	VAR robtarget OpenholeUD_4793 := [[479.2, -15.9, 180.72], [0.089899, 0.701369, 0.69888, -0.10755], [0,0,0,0], [9E9, 9E9, 9E9, 9E9, 9E9, 9E9]];
	VAR robtarget OpenholeUD_4794 := [[483.2, -15.9, 180.6], [0.102327, 0.699664, 0.696899, -0.119714], [0,0,0,0], [9E9, 9E9, 9E9, 9E9, 9E9, 9E9]];
	VAR robtarget OpenholeUD_4795 := [[487.2, -15.9, 180.48], [0.114451, 0.697783, 0.69476, -0.131563], [0,0,0,0], [9E9, 9E9, 9E9, 9E9, 9E9, 9E9]];
	VAR robtarget OpenholeUD_4796 := [[491.2, -15.9, 180.36], [0.126252, 0.695745, 0.69248, -0.143081], [0,0,0,0], [9E9, 9E9, 9E9, 9E9, 9E9, 9E9]];
	VAR robtarget OpenholeUD_4797 := [[495.19, -15.9, 180.24], [0.137713, 0.693567, 0.690077, -0.154251], [0,0,0,0], [9E9, 9E9, 9E9, 9E9, 9E9, 9E9]];
	VAR robtarget OpenholeUD_4798 := [[499.19, -15.9, 180.12], [0.148822, 0.691268, 0.687571, -0.165065], [0,0,0,0], [9E9, 9E9, 9E9, 9E9, 9E9, 9E9]];
	VAR robtarget OpenholeUD_4799 := [[503.19, -15.9, 180], [0.159571, 0.688867, 0.684978, -0.175514], [0,0,0,0], [9E9, 9E9, 9E9, 9E9, 9E9, 9E9]];
	VAR robtarget OpenholeUD_4800 := [[509.34, -15.9, 179.82], [0.183051, 0.683002, 0.683002, -0.183051], [0,0,0,0], [9E9, 9E9, 9E9, 9E9, 9E9, 9E9]];
	VAR robtarget OpenholeUD_4801 := [[513.34, -15.9, 179.8], [0.183051, 0.683002, 0.683002, -0.183051], [0,0,0,0], [9E9, 9E9, 9E9, 9E9, 9E9, 9E9]];
	VAR robtarget OpenholeUD_4802 := [[517.34, -15.9, 179.79], [0.183051, 0.683002, 0.683002, -0.183051], [0,0,0,0], [9E9, 9E9, 9E9, 9E9, 9E9, 9E9]];
	VAR robtarget OpenholeUD_4803 := [[521.34, -15.9, 179.78], [0.183051, 0.683002, 0.683002, -0.183051], [0,0,0,0], [9E9, 9E9, 9E9, 9E9, 9E9, 9E9]];
	VAR robtarget OpenholeUD_4804 := [[525.34, -15.9, 179.77], [0.183051, 0.683002, 0.683002, -0.183051], [0,0,0,0], [9E9, 9E9, 9E9, 9E9, 9E9, 9E9]];
	VAR robtarget OpenholeUD_4805 := [[529.34, -15.9, 179.75], [0.183051, 0.683002, 0.683002, -0.183051], [0,0,0,0], [9E9, 9E9, 9E9, 9E9, 9E9, 9E9]];
	VAR robtarget OpenholeUD_4806 := [[529.34, -15.9, 179.75], [0.183051, 0.683002, 0.683002, -0.183051], [0,0,0,0], [9E9, 9E9, 9E9, 9E9, 9E9, 9E9]];
	VAR robtarget OpenholeUD_4807 := [[529.34, -14.7, 179.06], [0.183051, 0.683002, 0.683002, -0.183051], [0,0,0,0], [9E9, 9E9, 9E9, 9E9, 9E9, 9E9]];
	VAR robtarget OpenholeUD_4808 := [[525.34, -14.7, 179.07], [0.183051, 0.683002, 0.683002, -0.183051], [0,0,0,0], [9E9, 9E9, 9E9, 9E9, 9E9, 9E9]];
	VAR robtarget OpenholeUD_4809 := [[521.34, -14.7, 179.09], [0.183051, 0.683002, 0.683002, -0.183051], [0,0,0,0], [9E9, 9E9, 9E9, 9E9, 9E9, 9E9]];
	VAR robtarget OpenholeUD_4810 := [[517.34, -14.7, 179.1], [0.183051, 0.683002, 0.683002, -0.183051], [0,0,0,0], [9E9, 9E9, 9E9, 9E9, 9E9, 9E9]];
	VAR robtarget OpenholeUD_4811 := [[513.34, -14.7, 179.11], [0.183051, 0.683002, 0.683002, -0.183051], [0,0,0,0], [9E9, 9E9, 9E9, 9E9, 9E9, 9E9]];
	VAR robtarget OpenholeUD_4812 := [[509.34, -14.7, 179.12], [0.183051, 0.683002, 0.683002, -0.183051], [0,0,0,0], [9E9, 9E9, 9E9, 9E9, 9E9, 9E9]];
	VAR robtarget OpenholeUD_4813 := [[505.34, -14.7, 179.29], [0.161707, 0.688368, 0.682625, -0.184452], [0,0,0,0], [9E9, 9E9, 9E9, 9E9, 9E9, 9E9]];
	VAR robtarget OpenholeUD_4814 := [[501.35, -14.7, 179.46], [0.15109, 0.690776, 0.685295, -0.174272], [0,0,0,0], [9E9, 9E9, 9E9, 9E9, 9E9, 9E9]];
	VAR robtarget OpenholeUD_4815 := [[497.35, -14.7, 179.62], [0.140112, 0.693086, 0.687891, -0.163724], [0,0,0,0], [9E9, 9E9, 9E9, 9E9, 9E9, 9E9]];
	VAR robtarget OpenholeUD_4816 := [[493.35, -14.7, 179.79], [0.12878, 0.695281, 0.690397, -0.152814], [0,0,0,0], [9E9, 9E9, 9E9, 9E9, 9E9, 9E9]];
	VAR robtarget OpenholeUD_4817 := [[489.36, -14.7, 179.96], [0.117104, 0.697343, 0.692794, -0.141548], [0,0,0,0], [9E9, 9E9, 9E9, 9E9, 9E9, 9E9]];
	VAR robtarget OpenholeUD_4818 := [[485.36, -14.7, 180.12], [0.105099, 0.699253, 0.695065, -0.129939], [0,0,0,0], [9E9, 9E9, 9E9, 9E9, 9E9, 9E9]];
	VAR robtarget OpenholeUD_4819 := [[481.36, -14.7, 180.29], [0.092784, 0.700993, 0.697191, -0.118001], [0,0,0,0], [9E9, 9E9, 9E9, 9E9, 9E9, 9E9]];
	VAR robtarget OpenholeUD_4820 := [[477.37, -14.7, 180.45], [0.08018, 0.702546, 0.699154, -0.105755], [0,0,0,0], [9E9, 9E9, 9E9, 9E9, 9E9, 9E9]];
	VAR robtarget OpenholeUD_4821 := [[473.37, -14.7, 180.62], [0.067317, 0.703895, 0.700935, -0.093223], [0,0,0,0], [9E9, 9E9, 9E9, 9E9, 9E9, 9E9]];
	VAR robtarget OpenholeUD_4822 := [[469.37, -14.7, 180.79], [0.054224, 0.705025, 0.702517, -0.080435], [0,0,0,0], [9E9, 9E9, 9E9, 9E9, 9E9, 9E9]];
	VAR robtarget OpenholeUD_4823 := [[465.38, -14.7, 180.95], [0.040937, 0.705921, 0.703885, -0.067421], [0,0,0,0], [9E9, 9E9, 9E9, 9E9, 9E9, 9E9]];
	VAR robtarget OpenholeUD_4824 := [[461.38, -14.7, 181.12], [0.027494, 0.706572, 0.705025, -0.054217], [0,0,0,0], [9E9, 9E9, 9E9, 9E9, 9E9, 9E9]];
	VAR robtarget OpenholeUD_4825 := [[454.47, -14.7, 181.41], [0.004004, 0.707095, 0.706425, -0.031051], [0,0,0,0], [9E9, 9E9, 9E9, 9E9, 9E9, 9E9]];
	VAR robtarget OpenholeUD_4826 := [[454.47, -14.7, 181.41], [0.004004, 0.707095, 0.706425, -0.031051], [0,0,0,0], [9E9, 9E9, 9E9, 9E9, 9E9, 9E9]];
	VAR robtarget OpenholeUD_4827 := [[453.25, -13.5, 181.41], [-0.004258, 0.707094, 0.706428, -0.030976], [0,0,0,0], [9E9, 9E9, 9E9, 9E9, 9E9, 9E9]];
	VAR robtarget OpenholeUD_4828 := [[457.24, -13.5, 181.2], [0.009373, 0.707045, 0.70571, -0.044424], [0,0,0,0], [9E9, 9E9, 9E9, 9E9, 9E9, 9E9]];
	VAR robtarget OpenholeUD_4829 := [[461.24, -13.5, 180.99], [0.022943, 0.706734, 0.704744, -0.057757], [0,0,0,0], [9E9, 9E9, 9E9, 9E9, 9E9, 9E9]];
	VAR robtarget OpenholeUD_4830 := [[465.23, -13.5, 180.78], [0.036407, 0.706169, 0.70354, -0.070934], [0,0,0,0], [9E9, 9E9, 9E9, 9E9, 9E9, 9E9]];
	VAR robtarget OpenholeUD_4831 := [[469.22, -13.5, 180.56], [0.049725, 0.705356, 0.70211, -0.083916], [0,0,0,0], [9E9, 9E9, 9E9, 9E9, 9E9, 9E9]];
	VAR robtarget OpenholeUD_4832 := [[473.22, -13.5, 180.35], [0.062857, 0.704307, 0.700468, -0.096668], [0,0,0,0], [9E9, 9E9, 9E9, 9E9, 9E9, 9E9]];
	VAR robtarget OpenholeUD_4833 := [[477.21, -13.5, 180.14], [0.075766, 0.703036, 0.69863, -0.109158], [0,0,0,0], [9E9, 9E9, 9E9, 9E9, 9E9, 9E9]];
	VAR robtarget OpenholeUD_4834 := [[481.21, -13.5, 179.93], [0.088422, 0.701557, 0.696615, -0.12136], [0,0,0,0], [9E9, 9E9, 9E9, 9E9, 9E9, 9E9]];
	VAR robtarget OpenholeUD_4835 := [[485.2, -13.5, 179.71], [0.100796, 0.699886, 0.694438, -0.13325], [0,0,0,0], [9E9, 9E9, 9E9, 9E9, 9E9, 9E9]];
	VAR robtarget OpenholeUD_4836 := [[489.2, -13.5, 179.5], [0.112865, 0.698041, 0.69212, -0.144808], [0,0,0,0], [9E9, 9E9, 9E9, 9E9, 9E9, 9E9]];
	VAR robtarget OpenholeUD_4837 := [[493.19, -13.5, 179.29], [0.124609, 0.696041, 0.689679, -0.15602], [0,0,0,0], [9E9, 9E9, 9E9, 9E9, 9E9, 9E9]];
	VAR robtarget OpenholeUD_4838 := [[497.18, -13.5, 179.08], [0.136013, 0.693902, 0.687134, -0.166875], [0,0,0,0], [9E9, 9E9, 9E9, 9E9, 9E9, 9E9]];
	VAR robtarget OpenholeUD_4839 := [[501.18, -13.5, 178.86], [0.147067, 0.691644, 0.684501, -0.177366], [0,0,0,0], [9E9, 9E9, 9E9, 9E9, 9E9, 9E9]];
	VAR robtarget OpenholeUD_4840 := [[505.17, -13.5, 178.65], [0.157761, 0.689283, 0.681798, -0.187488], [0,0,0,0], [9E9, 9E9, 9E9, 9E9, 9E9, 9E9]];
	VAR robtarget OpenholeUD_4841 := [[509.34, -13.5, 178.43], [0.183051, 0.683002, 0.683002, -0.183051], [0,0,0,0], [9E9, 9E9, 9E9, 9E9, 9E9, 9E9]];
	VAR robtarget OpenholeUD_4842 := [[513.34, -13.5, 178.42], [0.183051, 0.683002, 0.683002, -0.183051], [0,0,0,0], [9E9, 9E9, 9E9, 9E9, 9E9, 9E9]];
	VAR robtarget OpenholeUD_4843 := [[517.34, -13.5, 178.4], [0.183051, 0.683002, 0.683002, -0.183051], [0,0,0,0], [9E9, 9E9, 9E9, 9E9, 9E9, 9E9]];
	VAR robtarget OpenholeUD_4844 := [[521.34, -13.5, 178.39], [0.183051, 0.683002, 0.683002, -0.183051], [0,0,0,0], [9E9, 9E9, 9E9, 9E9, 9E9, 9E9]];
	VAR robtarget OpenholeUD_4845 := [[529.34, -13.5, 178.37], [0.183051, 0.683002, 0.683002, -0.183051], [0,0,0,0], [9E9, 9E9, 9E9, 9E9, 9E9, 9E9]];
	VAR robtarget OpenholeUD_4846 := [[529.34, -13.5, 178.37], [0.183051, 0.683002, 0.683002, -0.183051], [0,0,0,0], [9E9, 9E9, 9E9, 9E9, 9E9, 9E9]];
	VAR robtarget OpenholeUD_4847 := [[529.34, -12.3, 177.67], [0.183051, 0.683002, 0.683002, -0.183051], [0,0,0,0], [9E9, 9E9, 9E9, 9E9, 9E9, 9E9]];
	VAR robtarget OpenholeUD_4848 := [[525.34, -12.3, 177.69], [0.183051, 0.683002, 0.683002, -0.183051], [0,0,0,0], [9E9, 9E9, 9E9, 9E9, 9E9, 9E9]];
	VAR robtarget OpenholeUD_4849 := [[521.34, -12.3, 177.7], [0.183051, 0.683002, 0.683002, -0.183051], [0,0,0,0], [9E9, 9E9, 9E9, 9E9, 9E9, 9E9]];
	VAR robtarget OpenholeUD_4850 := [[517.34, -12.3, 177.71], [0.183051, 0.683002, 0.683002, -0.183051], [0,0,0,0], [9E9, 9E9, 9E9, 9E9, 9E9, 9E9]];
	VAR robtarget OpenholeUD_4851 := [[509.34, -12.3, 177.74], [0.183051, 0.683002, 0.683002, -0.183051], [0,0,0,0], [9E9, 9E9, 9E9, 9E9, 9E9, 9E9]];
	VAR robtarget OpenholeUD_4852 := [[505.34, -12.3, 178], [0.154707, 0.689975, 0.680721, -0.19136], [0,0,0,0], [9E9, 9E9, 9E9, 9E9, 9E9, 9E9]];
	VAR robtarget OpenholeUD_4853 := [[501.35, -12.3, 178.25], [0.143967, 0.692296, 0.683462, -0.181329], [0,0,0,0], [9E9, 9E9, 9E9, 9E9, 9E9, 9E9]];
	VAR robtarget OpenholeUD_4854 := [[497.36, -12.3, 178.51], [0.132871, 0.694511, 0.686137, -0.170928], [0,0,0,0], [9E9, 9E9, 9E9, 9E9, 9E9, 9E9]];
	VAR robtarget OpenholeUD_4855 := [[493.37, -12.3, 178.77], [0.121426, 0.696603, 0.68873, -0.16016], [0,0,0,0], [9E9, 9E9, 9E9, 9E9, 9E9, 9E9]];
	VAR robtarget OpenholeUD_4856 := [[489.38, -12.3, 179.03], [0.109644, 0.698554, 0.691223, -0.149033], [0,0,0,0], [9E9, 9E9, 9E9, 9E9, 9E9, 9E9]];
	VAR robtarget OpenholeUD_4857 := [[485.39, -12.3, 179.29], [0.09754, 0.700347, 0.693598, -0.137556], [0,0,0,0], [9E9, 9E9, 9E9, 9E9, 9E9, 9E9]];
	VAR robtarget OpenholeUD_4858 := [[481.39, -12.3, 179.55], [0.085135, 0.701963, 0.695837, -0.125744], [0,0,0,0], [9E9, 9E9, 9E9, 9E9, 9E9, 9E9]];
	VAR robtarget OpenholeUD_4859 := [[477.4, -12.3, 179.8], [0.072452, 0.703385, 0.69792, -0.113614], [0,0,0,0], [9E9, 9E9, 9E9, 9E9, 9E9, 9E9]];
	VAR robtarget OpenholeUD_4860 := [[473.41, -12.3, 180.06], [0.059519, 0.704597, 0.699829, -0.10119], [0,0,0,0], [9E9, 9E9, 9E9, 9E9, 9E9, 9E9]];
	VAR robtarget OpenholeUD_4861 := [[469.42, -12.3, 180.32], [0.046369, 0.705585, 0.701547, -0.088498], [0,0,0,0], [9E9, 9E9, 9E9, 9E9, 9E9, 9E9]];
	VAR robtarget OpenholeUD_4862 := [[465.43, -12.3, 180.58], [0.033038, 0.706335, 0.703057, -0.075569], [0,0,0,0], [9E9, 9E9, 9E9, 9E9, 9E9, 9E9]];
	VAR robtarget OpenholeUD_4863 := [[461.44, -12.3, 180.84], [0.019564, 0.706836, 0.704345, -0.062437], [0,0,0,0], [9E9, 9E9, 9E9, 9E9, 9E9, 9E9]];
	VAR robtarget OpenholeUD_4864 := [[457.44, -12.3, 181.1], [0.005991, 0.707081, 0.705397, -0.04914], [0,0,0,0], [9E9, 9E9, 9E9, 9E9, 9E9, 9E9]];
	VAR robtarget OpenholeUD_4865 := [[453.45, -12.3, 181.36], [-0.007638, 0.707066, 0.706204, -0.035718], [0,0,0,0], [9E9, 9E9, 9E9, 9E9, 9E9, 9E9]];
	VAR robtarget OpenholeUD_4866 := [[449.46, -12.3, 181.61], [-0.021278, 0.706787, 0.706758, -0.022215], [0,0,0,0], [9E9, 9E9, 9E9, 9E9, 9E9, 9E9]];
	VAR robtarget OpenholeUD_4867 := [[445.47, -12.3, 181.87], [-0.034882, 0.706246, 0.707054, -0.008673], [0,0,0,0], [9E9, 9E9, 9E9, 9E9, 9E9, 9E9]];
	VAR robtarget OpenholeUD_4868 := [[441.48, -12.3, 182.13], [-0.048405, 0.705448, 0.70709, 0.004862], [0,0,0,0], [9E9, 9E9, 9E9, 9E9, 9E9, 9E9]];
	VAR robtarget OpenholeUD_4869 := [[437.49, -12.3, 182.39], [-0.061804, 0.704401, 0.706869, 0.018346], [0,0,0,0], [9E9, 9E9, 9E9, 9E9, 9E9, 9E9]];
	VAR robtarget OpenholeUD_4870 := [[433.49, -12.3, 182.65], [-0.075036, 0.703114, 0.706394, 0.031737], [0,0,0,0], [9E9, 9E9, 9E9, 9E9, 9E9, 9E9]];
	VAR robtarget OpenholeUD_4871 := [[429.5, -12.3, 182.91], [-0.088063, 0.701602, 0.705674, 0.044994], [0,0,0,0], [9E9, 9E9, 9E9, 9E9, 9E9, 9E9]];
	VAR robtarget OpenholeUD_4872 := [[425.51, -12.3, 183.16], [-0.100848, 0.699878, 0.704718, 0.058077], [0,0,0,0], [9E9, 9E9, 9E9, 9E9, 9E9, 9E9]];
	VAR robtarget OpenholeUD_4873 := [[421.52, -12.3, 183.42], [-0.11336, 0.697961, 0.703538, 0.070951], [0,0,0,0], [9E9, 9E9, 9E9, 9E9, 9E9, 9E9]];
	VAR robtarget OpenholeUD_4874 := [[417.53, -12.3, 183.68], [-0.125573, 0.695867, 0.702149, 0.083585], [0,0,0,0], [9E9, 9E9, 9E9, 9E9, 9E9, 9E9]];
	VAR robtarget OpenholeUD_4875 := [[413.54, -12.3, 183.94], [-0.137462, 0.693617, 0.700567, 0.095951], [0,0,0,0], [9E9, 9E9, 9E9, 9E9, 9E9, 9E9]];
	VAR robtarget OpenholeUD_4876 := [[409.54, -12.3, 184.2], [-0.149009, 0.691228, 0.698807, 0.108023], [0,0,0,0], [9E9, 9E9, 9E9, 9E9, 9E9, 9E9]];
	VAR robtarget OpenholeUD_4877 := [[405.55, -12.3, 184.46], [-0.1602, 0.688721, 0.696887, 0.119783], [0,0,0,0], [9E9, 9E9, 9E9, 9E9, 9E9, 9E9]];
	VAR robtarget OpenholeUD_4878 := [[401.56, -12.3, 184.72], [-0.171025, 0.686113, 0.694826, 0.131214], [0,0,0,0], [9E9, 9E9, 9E9, 9E9, 9E9, 9E9]];
	VAR robtarget OpenholeUD_4879 := [[397.57, -12.3, 184.97], [-0.181476, 0.683423, 0.69264, 0.142304], [0,0,0,0], [9E9, 9E9, 9E9, 9E9, 9E9, 9E9]];
	VAR robtarget OpenholeUD_4880 := [[393.58, -12.3, 185.23], [-0.191552, 0.680667, 0.690346, 0.153045], [0,0,0,0], [9E9, 9E9, 9E9, 9E9, 9E9, 9E9]];
	VAR robtarget OpenholeUD_4881 := [[389.36, -12.3, 185.51], [-0.201793, 0.677702, 0.687823, 0.164011], [0,0,0,0], [9E9, 9E9, 9E9, 9E9, 9E9, 9E9]];
	VAR robtarget OpenholeUD_4882 := [[385.36, -12.3, 185.52], [-0.183051, 0.683002, 0.683002, 0.183051], [0,0,0,0], [9E9, 9E9, 9E9, 9E9, 9E9, 9E9]];
	VAR robtarget OpenholeUD_4883 := [[381.36, -12.3, 185.53], [-0.183051, 0.683002, 0.683002, 0.183051], [0,0,0,0], [9E9, 9E9, 9E9, 9E9, 9E9, 9E9]];
	VAR robtarget OpenholeUD_4884 := [[377.36, -12.3, 185.54], [-0.183051, 0.683002, 0.683002, 0.183051], [0,0,0,0], [9E9, 9E9, 9E9, 9E9, 9E9, 9E9]];
	VAR robtarget OpenholeUD_4885 := [[373.36, -12.3, 185.56], [-0.183051, 0.683002, 0.683002, 0.183051], [0,0,0,0], [9E9, 9E9, 9E9, 9E9, 9E9, 9E9]];
	VAR robtarget OpenholeUD_4886 := [[369.36, -12.3, 185.57], [-0.183051, 0.683002, 0.683002, 0.183051], [0,0,0,0], [9E9, 9E9, 9E9, 9E9, 9E9, 9E9]];
	VAR robtarget OpenholeUD_4887 := [[369.36, -12.3, 185.57], [-0.183051, 0.683002, 0.683002, 0.183051], [0,0,0,0], [9E9, 9E9, 9E9, 9E9, 9E9, 9E9]];
	VAR robtarget OpenholeUD_4888 := [[369.36, -13.5, 184.88], [-0.183051, 0.683002, 0.683002, 0.183051], [0,0,0,0], [9E9, 9E9, 9E9, 9E9, 9E9, 9E9]];
	VAR robtarget OpenholeUD_4889 := [[373.36, -13.5, 184.86], [-0.183051, 0.683002, 0.683002, 0.183051], [0,0,0,0], [9E9, 9E9, 9E9, 9E9, 9E9, 9E9]];
	VAR robtarget OpenholeUD_4890 := [[377.36, -13.5, 184.85], [-0.183051, 0.683002, 0.683002, 0.183051], [0,0,0,0], [9E9, 9E9, 9E9, 9E9, 9E9, 9E9]];
	VAR robtarget OpenholeUD_4891 := [[381.36, -13.5, 184.84], [-0.183051, 0.683002, 0.683002, 0.183051], [0,0,0,0], [9E9, 9E9, 9E9, 9E9, 9E9, 9E9]];
	VAR robtarget OpenholeUD_4892 := [[389.36, -13.5, 184.81], [-0.198402, 0.678702, 0.686998, 0.167434], [0,0,0,0], [9E9, 9E9, 9E9, 9E9, 9E9, 9E9]];
	VAR robtarget OpenholeUD_4893 := [[393.35, -13.5, 184.6], [-0.188647, 0.681478, 0.689428, 0.157129], [0,0,0,0], [9E9, 9E9, 9E9, 9E9, 9E9, 9E9]];
	VAR robtarget OpenholeUD_4894 := [[397.35, -13.5, 184.39], [-0.178516, 0.684202, 0.691771, 0.146467], [0,0,0,0], [9E9, 9E9, 9E9, 9E9, 9E9, 9E9]];
	VAR robtarget OpenholeUD_4895 := [[401.34, -13.5, 184.18], [-0.168011, 0.686857, 0.694012, 0.135454], [0,0,0,0], [9E9, 9E9, 9E9, 9E9, 9E9, 9E9]];
	VAR robtarget OpenholeUD_4896 := [[405.33, -13.5, 183.96], [-0.157134, 0.689427, 0.696132, 0.124096], [0,0,0,0], [9E9, 9E9, 9E9, 9E9, 9E9, 9E9]];
	VAR robtarget OpenholeUD_4897 := [[409.33, -13.5, 183.75], [-0.145892, 0.691893, 0.698115, 0.112405], [0,0,0,0], [9E9, 9E9, 9E9, 9E9, 9E9, 9E9]];
	VAR robtarget OpenholeUD_4898 := [[413.32, -13.5, 183.54], [-0.134296, 0.694237, 0.699943, 0.100396], [0,0,0,0], [9E9, 9E9, 9E9, 9E9, 9E9, 9E9]];
	VAR robtarget OpenholeUD_4899 := [[417.32, -13.5, 183.33], [-0.122361, 0.696439, 0.701598, 0.08809], [0,0,0,0], [9E9, 9E9, 9E9, 9E9, 9E9, 9E9]];
	VAR robtarget OpenholeUD_4900 := [[421.31, -13.5, 183.11], [-0.110106, 0.698482, 0.703064, 0.075508], [0,0,0,0], [9E9, 9E9, 9E9, 9E9, 9E9, 9E9]];
	VAR robtarget OpenholeUD_4901 := [[425.31, -13.5, 182.9], [-0.097554, 0.700345, 0.704323, 0.062679], [0,0,0,0], [9E9, 9E9, 9E9, 9E9, 9E9, 9E9]];
	VAR robtarget OpenholeUD_4902 := [[429.3, -13.5, 182.69], [-0.084733, 0.702012, 0.705363, 0.049633], [0,0,0,0], [9E9, 9E9, 9E9, 9E9, 9E9, 9E9]];
	VAR robtarget OpenholeUD_4903 := [[433.29, -13.5, 182.48], [-0.071675, 0.703465, 0.706169, 0.036405], [0,0,0,0], [9E9, 9E9, 9E9, 9E9, 9E9, 9E9]];
	VAR robtarget OpenholeUD_4904 := [[437.29, -13.5, 182.26], [-0.058416, 0.70469, 0.706731, 0.023035], [0,0,0,0], [9E9, 9E9, 9E9, 9E9, 9E9, 9E9]];
	VAR robtarget OpenholeUD_4905 := [[441.28, -13.5, 182.05], [-0.044995, 0.705674, 0.707042, 0.009561], [0,0,0,0], [9E9, 9E9, 9E9, 9E9, 9E9, 9E9]];
	VAR robtarget OpenholeUD_4906 := [[445.45, -13.5, 181.83], [-0.030877, 0.706432, 0.707092, -0.004547], [0,0,0,0], [9E9, 9E9, 9E9, 9E9, 9E9, 9E9]];
	VAR robtarget OpenholeUD_4907 := [[445.45, -13.5, 181.83], [-0.030877, 0.706432, 0.707092, -0.004547], [0,0,0,0], [9E9, 9E9, 9E9, 9E9, 9E9, 9E9]];
	VAR robtarget OpenholeUD_4908 := [[444.22, -14.7, 181.83], [-0.030953, 0.706429, 0.707097, 0.003656], [0,0,0,0], [9E9, 9E9, 9E9, 9E9, 9E9, 9E9]];
	VAR robtarget OpenholeUD_4909 := [[440.23, -14.7, 182], [-0.044489, 0.705706, 0.706898, 0.017174], [0,0,0,0], [9E9, 9E9, 9E9, 9E9, 9E9, 9E9]];
	VAR robtarget OpenholeUD_4910 := [[436.23, -14.7, 182.17], [-0.0579, 0.704732, 0.706444, 0.030612], [0,0,0,0], [9E9, 9E9, 9E9, 9E9, 9E9, 9E9]];
	VAR robtarget OpenholeUD_4911 := [[432.23, -14.7, 182.33], [-0.071146, 0.703518, 0.705741, 0.04393], [0,0,0,0], [9E9, 9E9, 9E9, 9E9, 9E9, 9E9]];
	VAR robtarget OpenholeUD_4912 := [[428.24, -14.7, 182.5], [-0.084187, 0.702077, 0.704799, 0.057088], [0,0,0,0], [9E9, 9E9, 9E9, 9E9, 9E9, 9E9]];
	VAR robtarget OpenholeUD_4913 := [[424.24, -14.7, 182.67], [-0.096988, 0.700424, 0.703629, 0.070048], [0,0,0,0], [9E9, 9E9, 9E9, 9E9, 9E9, 9E9]];
	VAR robtarget OpenholeUD_4914 := [[420.25, -14.7, 182.83], [-0.109517, 0.698574, 0.702245, 0.082777], [0,0,0,0], [9E9, 9E9, 9E9, 9E9, 9E9, 9E9]];
	VAR robtarget OpenholeUD_4915 := [[416.25, -14.7, 183], [-0.121748, 0.696547, 0.700663, 0.095245], [0,0,0,0], [9E9, 9E9, 9E9, 9E9, 9E9, 9E9]];
	VAR robtarget OpenholeUD_4916 := [[412.25, -14.7, 183.17], [-0.133657, 0.69436, 0.698899, 0.107427], [0,0,0,0], [9E9, 9E9, 9E9, 9E9, 9E9, 9E9]];
	VAR robtarget OpenholeUD_4917 := [[408.26, -14.7, 183.33], [-0.145225, 0.692033, 0.69697, 0.119301], [0,0,0,0], [9E9, 9E9, 9E9, 9E9, 9E9, 9E9]];
	VAR robtarget OpenholeUD_4918 := [[404.26, -14.7, 183.5], [-0.15644, 0.689584, 0.694895, 0.13085], [0,0,0,0], [9E9, 9E9, 9E9, 9E9, 9E9, 9E9]];
	VAR robtarget OpenholeUD_4919 := [[400.26, -14.7, 183.67], [-0.167289, 0.687033, 0.69269, 0.142058], [0,0,0,0], [9E9, 9E9, 9E9, 9E9, 9E9, 9E9]];
	VAR robtarget OpenholeUD_4920 := [[396.27, -14.7, 183.83], [-0.177767, 0.684397, 0.690374, 0.152918], [0,0,0,0], [9E9, 9E9, 9E9, 9E9, 9E9, 9E9]];
	VAR robtarget OpenholeUD_4921 := [[389.35, -14.7, 184.12], [-0.195004, 0.679686, 0.686155, 0.170856], [0,0,0,0], [9E9, 9E9, 9E9, 9E9, 9E9, 9E9]];
	VAR robtarget OpenholeUD_4922 := [[385.35, -14.7, 184.13], [-0.183051, 0.683002, 0.683002, 0.183051], [0,0,0,0], [9E9, 9E9, 9E9, 9E9, 9E9, 9E9]];
	VAR robtarget OpenholeUD_4923 := [[381.35, -14.7, 184.15], [-0.183051, 0.683002, 0.683002, 0.183051], [0,0,0,0], [9E9, 9E9, 9E9, 9E9, 9E9, 9E9]];
	VAR robtarget OpenholeUD_4924 := [[377.35, -14.7, 184.16], [-0.183051, 0.683002, 0.683002, 0.183051], [0,0,0,0], [9E9, 9E9, 9E9, 9E9, 9E9, 9E9]];
	VAR robtarget OpenholeUD_4925 := [[369.35, -14.7, 184.18], [-0.183051, 0.683002, 0.683002, 0.183051], [0,0,0,0], [9E9, 9E9, 9E9, 9E9, 9E9, 9E9]];
	VAR robtarget OpenholeUD_4926 := [[369.35, -14.7, 184.18], [-0.183051, 0.683002, 0.683002, 0.183051], [0,0,0,0], [9E9, 9E9, 9E9, 9E9, 9E9, 9E9]];
	VAR robtarget OpenholeUD_4927 := [[369.35, -15.9, 183.49], [-0.183051, 0.683002, 0.683002, 0.183051], [0,0,0,0], [9E9, 9E9, 9E9, 9E9, 9E9, 9E9]];
	VAR robtarget OpenholeUD_4928 := [[373.35, -15.9, 183.48], [-0.183051, 0.683002, 0.683002, 0.183051], [0,0,0,0], [9E9, 9E9, 9E9, 9E9, 9E9, 9E9]];
	VAR robtarget OpenholeUD_4929 := [[377.35, -15.9, 183.46], [-0.183051, 0.683002, 0.683002, 0.183051], [0,0,0,0], [9E9, 9E9, 9E9, 9E9, 9E9, 9E9]];
	VAR robtarget OpenholeUD_4930 := [[381.35, -15.9, 183.45], [-0.183051, 0.683002, 0.683002, 0.183051], [0,0,0,0], [9E9, 9E9, 9E9, 9E9, 9E9, 9E9]];
	VAR robtarget OpenholeUD_4931 := [[389.35, -15.9, 183.43], [-0.191598, 0.680654, 0.685294, 0.174276], [0,0,0,0], [9E9, 9E9, 9E9, 9E9, 9E9, 9E9]];
	VAR robtarget OpenholeUD_4932 := [[393.35, -15.9, 183.31], [-0.181693, 0.683365, 0.687802, 0.164098], [0,0,0,0], [9E9, 9E9, 9E9, 9E9, 9E9, 9E9]];
	VAR robtarget OpenholeUD_4933 := [[397.35, -15.9, 183.19], [-0.171414, 0.686016, 0.690231, 0.153561], [0,0,0,0], [9E9, 9E9, 9E9, 9E9, 9E9, 9E9]];
	VAR robtarget OpenholeUD_4934 := [[401.35, -15.9, 183.07], [-0.160762, 0.688589, 0.692565, 0.142666], [0,0,0,0], [9E9, 9E9, 9E9, 9E9, 9E9, 9E9]];
	VAR robtarget OpenholeUD_4935 := [[405.35, -15.9, 182.95], [-0.149743, 0.691069, 0.694786, 0.131423], [0,0,0,0], [9E9, 9E9, 9E9, 9E9, 9E9, 9E9]];
	VAR robtarget OpenholeUD_4936 := [[409.34, -15.9, 182.83], [-0.138364, 0.693437, 0.696878, 0.11984], [0,0,0,0], [9E9, 9E9, 9E9, 9E9, 9E9, 9E9]];
	VAR robtarget OpenholeUD_4937 := [[413.34, -15.9, 182.7], [-0.126637, 0.695675, 0.698821, 0.107932], [0,0,0,0], [9E9, 9E9, 9E9, 9E9, 9E9, 9E9]];
	VAR robtarget OpenholeUD_4938 := [[417.34, -15.9, 182.58], [-0.114578, 0.697762, 0.700599, 0.095717], [0,0,0,0], [9E9, 9E9, 9E9, 9E9, 9E9, 9E9]];
	VAR robtarget OpenholeUD_4939 := [[421.34, -15.9, 182.46], [-0.102208, 0.699681, 0.702193, 0.083217], [0,0,0,0], [9E9, 9E9, 9E9, 9E9, 9E9, 9E9]];
	VAR robtarget OpenholeUD_4940 := [[425.34, -15.9, 182.34], [-0.08955, 0.701413, 0.703588, 0.07046], [0,0,0,0], [9E9, 9E9, 9E9, 9E9, 9E9, 9E9]];
	VAR robtarget OpenholeUD_4941 := [[429.33, -15.9, 182.22], [-0.076635, 0.702942, 0.704767, 0.057474], [0,0,0,0], [9E9, 9E9, 9E9, 9E9, 9E9, 9E9]];
	VAR robtarget OpenholeUD_4942 := [[433.33, -15.9, 182.1], [-0.063495, 0.70425, 0.705718, 0.044294], [0,0,0,0], [9E9, 9E9, 9E9, 9E9, 9E9, 9E9]];
	VAR robtarget OpenholeUD_4943 := [[437.33, -15.9, 181.98], [-0.050168, 0.705325, 0.706429, 0.030958], [0,0,0,0], [9E9, 9E9, 9E9, 9E9, 9E9, 9E9]];
	VAR robtarget OpenholeUD_4944 := [[443.48, -15.9, 181.8], [-0.029392, 0.706496, 0.707033, 0.010229], [0,0,0,0], [9E9, 9E9, 9E9, 9E9, 9E9, 9E9]];
	VAR robtarget OpenholeUD_4945 := [[443.48, -15.9, 181.8], [-0.029392, 0.706496, 0.707033, 0.010229], [0,0,0,0], [9E9, 9E9, 9E9, 9E9, 9E9, 9E9]];
	VAR robtarget OpenholeUD_4946 := [[443.05, -17.1, 181.74], [-0.02678, 0.706599, 0.706931, 0.015756], [0,0,0,0], [9E9, 9E9, 9E9, 9E9, 9E9, 9E9]];
	VAR robtarget OpenholeUD_4947 := [[439.05, -17.1, 181.81], [-0.040325, 0.705956, 0.706502, 0.029235], [0,0,0,0], [9E9, 9E9, 9E9, 9E9, 9E9, 9E9]];
	VAR robtarget OpenholeUD_4948 := [[435.05, -17.1, 181.89], [-0.053748, 0.705061, 0.705822, 0.042608], [0,0,0,0], [9E9, 9E9, 9E9, 9E9, 9E9, 9E9]];
	VAR robtarget OpenholeUD_4949 := [[431.05, -17.1, 181.96], [-0.067007, 0.703925, 0.704899, 0.055835], [0,0,0,0], [9E9, 9E9, 9E9, 9E9, 9E9, 9E9]];
	VAR robtarget OpenholeUD_4950 := [[427.05, -17.1, 182.03], [-0.080063, 0.70256, 0.703744, 0.068876], [0,0,0,0], [9E9, 9E9, 9E9, 9E9, 9E9, 9E9]];
	VAR robtarget OpenholeUD_4951 := [[423.05, -17.1, 182.11], [-0.092881, 0.70098, 0.702371, 0.081698], [0,0,0,0], [9E9, 9E9, 9E9, 9E9, 9E9, 9E9]];
	VAR robtarget OpenholeUD_4952 := [[419.05, -17.1, 182.18], [-0.10543, 0.699203, 0.700795, 0.094269], [0,0,0,0], [9E9, 9E9, 9E9, 9E9, 9E9, 9E9]];
	VAR robtarget OpenholeUD_4953 := [[415.05, -17.1, 182.26], [-0.117681, 0.697245, 0.699031, 0.106561], [0,0,0,0], [9E9, 9E9, 9E9, 9E9, 9E9, 9E9]];
	VAR robtarget OpenholeUD_4954 := [[411.05, -17.1, 182.33], [-0.129613, 0.695126, 0.697098, 0.11855], [0,0,0,0], [9E9, 9E9, 9E9, 9E9, 9E9, 9E9]];
	VAR robtarget OpenholeUD_4955 := [[407.05, -17.1, 182.41], [-0.141207, 0.692864, 0.695013, 0.130218], [0,0,0,0], [9E9, 9E9, 9E9, 9E9, 9E9, 9E9]];
	VAR robtarget OpenholeUD_4956 := [[403.05, -17.1, 182.48], [-0.152448, 0.690478, 0.692794, 0.141549], [0,0,0,0], [9E9, 9E9, 9E9, 9E9, 9E9, 9E9]];
	VAR robtarget OpenholeUD_4957 := [[399.06, -17.1, 182.55], [-0.163327, 0.687986, 0.690459, 0.152532], [0,0,0,0], [9E9, 9E9, 9E9, 9E9, 9E9, 9E9]];
	VAR robtarget OpenholeUD_4958 := [[395.06, -17.1, 182.63], [-0.173837, 0.685406, 0.688026, 0.163159], [0,0,0,0], [9E9, 9E9, 9E9, 9E9, 9E9, 9E9]];
	VAR robtarget OpenholeUD_4959 := [[389.35, -17.1, 182.73], [-0.188186, 0.681606, 0.684416, 0.177694], [0,0,0,0], [9E9, 9E9, 9E9, 9E9, 9E9, 9E9]];
	VAR robtarget OpenholeUD_4960 := [[385.35, -17.1, 182.75], [-0.183051, 0.683002, 0.683002, 0.183051], [0,0,0,0], [9E9, 9E9, 9E9, 9E9, 9E9, 9E9]];
	VAR robtarget OpenholeUD_4961 := [[381.35, -17.1, 182.76], [-0.183051, 0.683002, 0.683002, 0.183051], [0,0,0,0], [9E9, 9E9, 9E9, 9E9, 9E9, 9E9]];
	VAR robtarget OpenholeUD_4962 := [[377.35, -17.1, 182.77], [-0.183051, 0.683002, 0.683002, 0.183051], [0,0,0,0], [9E9, 9E9, 9E9, 9E9, 9E9, 9E9]];
	VAR robtarget OpenholeUD_4963 := [[369.35, -17.1, 182.8], [-0.183051, 0.683002, 0.683002, 0.183051], [0,0,0,0], [9E9, 9E9, 9E9, 9E9, 9E9, 9E9]];
	VAR robtarget OpenholeUD_4964 := [[369.35, -17.1, 182.8], [-0.183051, 0.683002, 0.683002, 0.183051], [0,0,0,0], [9E9, 9E9, 9E9, 9E9, 9E9, 9E9]];
	VAR robtarget OpenholeUD_4965 := [[369.35, -18.3, 182.1], [-0.183051, 0.683002, 0.683002, 0.183051], [0,0,0,0], [9E9, 9E9, 9E9, 9E9, 9E9, 9E9]];
	VAR robtarget OpenholeUD_4966 := [[373.35, -18.3, 182.09], [-0.183051, 0.683002, 0.683002, 0.183051], [0,0,0,0], [9E9, 9E9, 9E9, 9E9, 9E9, 9E9]];
	VAR robtarget OpenholeUD_4967 := [[377.35, -18.3, 182.08], [-0.183051, 0.683002, 0.683002, 0.183051], [0,0,0,0], [9E9, 9E9, 9E9, 9E9, 9E9, 9E9]];
	VAR robtarget OpenholeUD_4968 := [[381.35, -18.3, 182.07], [-0.183051, 0.683002, 0.683002, 0.183051], [0,0,0,0], [9E9, 9E9, 9E9, 9E9, 9E9, 9E9]];
	VAR robtarget OpenholeUD_4969 := [[385.35, -18.3, 182.05], [-0.183051, 0.683002, 0.683002, 0.183051], [0,0,0,0], [9E9, 9E9, 9E9, 9E9, 9E9, 9E9]];
	VAR robtarget OpenholeUD_4970 := [[389.35, -18.3, 182.04], [-0.184767, 0.68254, 0.68352, 0.181109], [0,0,0,0], [9E9, 9E9, 9E9, 9E9, 9E9, 9E9]];
	VAR robtarget OpenholeUD_4971 := [[393.35, -18.3, 182.01], [-0.174717, 0.685182, 0.686103, 0.171065], [0,0,0,0], [9E9, 9E9, 9E9, 9E9, 9E9, 9E9]];
	VAR robtarget OpenholeUD_4972 := [[397.35, -18.3, 181.98], [-0.164295, 0.687755, 0.688614, 0.160658], [0,0,0,0], [9E9, 9E9, 9E9, 9E9, 9E9, 9E9]];
	VAR robtarget OpenholeUD_4973 := [[401.35, -18.3, 181.96], [-0.153504, 0.690244, 0.691038, 0.14989], [0,0,0,0], [9E9, 9E9, 9E9, 9E9, 9E9, 9E9]];
	VAR robtarget OpenholeUD_4974 := [[405.35, -18.3, 181.93], [-0.14235, 0.69263, 0.693356, 0.138769], [0,0,0,0], [9E9, 9E9, 9E9, 9E9, 9E9, 9E9]];
	VAR robtarget OpenholeUD_4975 := [[409.35, -18.3, 181.9], [-0.130841, 0.694896, 0.695553, 0.127302], [0,0,0,0], [9E9, 9E9, 9E9, 9E9, 9E9, 9E9]];
	VAR robtarget OpenholeUD_4976 := [[413.35, -18.3, 181.87], [-0.11899, 0.697023, 0.697609, 0.115503], [0,0,0,0], [9E9, 9E9, 9E9, 9E9, 9E9, 9E9]];
	VAR robtarget OpenholeUD_4977 := [[417.35, -18.3, 181.85], [-0.106816, 0.698992, 0.699507, 0.103389], [0,0,0,0], [9E9, 9E9, 9E9, 9E9, 9E9, 9E9]];
	VAR robtarget OpenholeUD_4978 := [[421.35, -18.3, 181.82], [-0.094339, 0.700785, 0.701229, 0.090981], [0,0,0,0], [9E9, 9E9, 9E9, 9E9, 9E9, 9E9]];
	VAR robtarget OpenholeUD_4979 := [[425.35, -18.3, 181.79], [-0.081585, 0.702384, 0.702758, 0.078305], [0,0,0,0], [9E9, 9E9, 9E9, 9E9, 9E9, 9E9]];
	VAR robtarget OpenholeUD_4980 := [[429.35, -18.3, 181.76], [-0.068586, 0.703773, 0.704077, 0.065389], [0,0,0,0], [9E9, 9E9, 9E9, 9E9, 9E9, 9E9]];
	VAR robtarget OpenholeUD_4981 := [[433.35, -18.3, 181.73], [-0.055374, 0.704935, 0.705172, 0.052266], [0,0,0,0], [9E9, 9E9, 9E9, 9E9, 9E9, 9E9]];
	VAR robtarget OpenholeUD_4982 := [[437.35, -18.3, 181.71], [-0.041988, 0.705859, 0.706032, 0.038974], [0,0,0,0], [9E9, 9E9, 9E9, 9E9, 9E9, 9E9]];
	VAR robtarget OpenholeUD_4983 := [[442.86, -18.3, 181.67], [-0.02333, 0.706722, 0.706811, 0.02045], [0,0,0,0], [9E9, 9E9, 9E9, 9E9, 9E9, 9E9]];
	VAR robtarget OpenholeUD_4984 := [[442.86, -18.3, 181.67], [-0.02333, 0.706722, 0.706811, 0.02045], [0,0,0,0], [9E9, 9E9, 9E9, 9E9, 9E9, 9E9]];
	VAR robtarget OpenholeUD_4985 := [[442.9, -19.5, 181.59], [-0.019116, 0.706848, 0.706686, 0.024384], [0,0,0,0], [9E9, 9E9, 9E9, 9E9, 9E9, 9E9]];
	VAR robtarget OpenholeUD_4986 := [[438.9, -19.5, 181.57], [-0.03269, 0.706351, 0.706094, 0.03783], [0,0,0,0], [9E9, 9E9, 9E9, 9E9, 9E9, 9E9]];
	VAR robtarget OpenholeUD_4987 := [[434.9, -19.5, 181.56], [-0.046156, 0.705599, 0.705254, 0.051155], [0,0,0,0], [9E9, 9E9, 9E9, 9E9, 9E9, 9E9]];
	VAR robtarget OpenholeUD_4988 := [[430.9, -19.5, 181.54], [-0.059469, 0.704602, 0.704176, 0.064318], [0,0,0,0], [9E9, 9E9, 9E9, 9E9, 9E9, 9E9]];
	VAR robtarget OpenholeUD_4989 := [[426.9, -19.5, 181.52], [-0.072592, 0.703371, 0.702871, 0.077282], [0,0,0,0], [9E9, 9E9, 9E9, 9E9, 9E9, 9E9]];
	VAR robtarget OpenholeUD_4990 := [[422.9, -19.5, 181.5], [-0.085487, 0.70192, 0.701354, 0.090014], [0,0,0,0], [9E9, 9E9, 9E9, 9E9, 9E9, 9E9]];
	VAR robtarget OpenholeUD_4991 := [[418.9, -19.5, 181.48], [-0.098122, 0.700266, 0.699641, 0.102482], [0,0,0,0], [9E9, 9E9, 9E9, 9E9, 9E9, 9E9]];
	VAR robtarget OpenholeUD_4992 := [[414.9, -19.5, 181.46], [-0.11047, 0.698424, 0.697749, 0.11466], [0,0,0,0], [9E9, 9E9, 9E9, 9E9, 9E9, 9E9]];
	VAR robtarget OpenholeUD_4993 := [[410.9, -19.5, 181.45], [-0.122505, 0.696414, 0.695695, 0.126527], [0,0,0,0], [9E9, 9E9, 9E9, 9E9, 9E9, 9E9]];
	VAR robtarget OpenholeUD_4994 := [[406.9, -19.5, 181.43], [-0.134209, 0.694253, 0.693497, 0.138065], [0,0,0,0], [9E9, 9E9, 9E9, 9E9, 9E9, 9E9]];
	VAR robtarget OpenholeUD_4995 := [[402.9, -19.5, 181.41], [-0.145566, 0.691961, 0.691174, 0.149259], [0,0,0,0], [9E9, 9E9, 9E9, 9E9, 9E9, 9E9]];
	VAR robtarget OpenholeUD_4996 := [[398.9, -19.5, 181.39], [-0.156566, 0.689556, 0.688744, 0.160099], [0,0,0,0], [9E9, 9E9, 9E9, 9E9, 9E9, 9E9]];
	VAR robtarget OpenholeUD_4997 := [[394.9, -19.5, 181.37], [-0.167199, 0.687055, 0.686224, 0.170579], [0,0,0,0], [9E9, 9E9, 9E9, 9E9, 9E9, 9E9]];
	VAR robtarget OpenholeUD_4998 := [[389.35, -19.5, 181.35], [-0.181344, 0.683458, 0.682607, 0.18452], [0,0,0,0], [9E9, 9E9, 9E9, 9E9, 9E9, 9E9]];
	VAR robtarget OpenholeUD_4999 := [[385.35, -19.5, 181.36], [-0.183051, 0.683002, 0.683002, 0.183051], [0,0,0,0], [9E9, 9E9, 9E9, 9E9, 9E9, 9E9]];
	VAR robtarget OpenholeUD_5000 := [[381.35, -19.5, 181.37], [-0.183051, 0.683002, 0.683002, 0.183051], [0,0,0,0], [9E9, 9E9, 9E9, 9E9, 9E9, 9E9]];
	VAR robtarget OpenholeUD_5001 := [[377.35, -19.5, 181.39], [-0.183051, 0.683002, 0.683002, 0.183051], [0,0,0,0], [9E9, 9E9, 9E9, 9E9, 9E9, 9E9]];
	VAR robtarget OpenholeUD_5002 := [[373.35, -19.5, 181.4], [-0.183051, 0.683002, 0.683002, 0.183051], [0,0,0,0], [9E9, 9E9, 9E9, 9E9, 9E9, 9E9]];
	VAR robtarget OpenholeUD_5003 := [[369.35, -19.5, 181.41], [-0.183051, 0.683002, 0.683002, 0.183051], [0,0,0,0], [9E9, 9E9, 9E9, 9E9, 9E9, 9E9]];
	VAR robtarget OpenholeUD_5004 := [[369.35, -19.5, 181.41], [-0.183051, 0.683002, 0.683002, 0.183051], [0,0,0,0], [9E9, 9E9, 9E9, 9E9, 9E9, 9E9]];
	VAR robtarget OpenholeUD_5005 := [[369.34, -20.7, 180.72], [-0.183051, 0.683002, 0.683002, 0.183051], [0,0,0,0], [9E9, 9E9, 9E9, 9E9, 9E9, 9E9]];
	VAR robtarget OpenholeUD_5006 := [[373.34, -20.7, 180.71], [-0.183051, 0.683002, 0.683002, 0.183051], [0,0,0,0], [9E9, 9E9, 9E9, 9E9, 9E9, 9E9]];
	VAR robtarget OpenholeUD_5007 := [[377.34, -20.7, 180.69], [-0.183051, 0.683002, 0.683002, 0.183051], [0,0,0,0], [9E9, 9E9, 9E9, 9E9, 9E9, 9E9]];
	VAR robtarget OpenholeUD_5008 := [[381.34, -20.7, 180.68], [-0.183051, 0.683002, 0.683002, 0.183051], [0,0,0,0], [9E9, 9E9, 9E9, 9E9, 9E9, 9E9]];
	VAR robtarget OpenholeUD_5009 := [[385.34, -20.7, 180.67], [-0.183051, 0.683002, 0.683002, 0.183051], [0,0,0,0], [9E9, 9E9, 9E9, 9E9, 9E9, 9E9]];
	VAR robtarget OpenholeUD_5010 := [[389.34, -20.7, 180.65], [-0.177916, 0.684358, 0.681677, 0.187926], [0,0,0,0], [9E9, 9E9, 9E9, 9E9, 9E9, 9E9]];
	VAR robtarget OpenholeUD_5011 := [[393.34, -20.7, 180.72], [-0.167726, 0.686926, 0.684331, 0.178021], [0,0,0,0], [9E9, 9E9, 9E9, 9E9, 9E9, 9E9]];
	VAR robtarget OpenholeUD_5012 := [[397.34, -20.7, 180.78], [-0.157168, 0.689419, 0.68692, 0.167751], [0,0,0,0], [9E9, 9E9, 9E9, 9E9, 9E9, 9E9]];
	VAR robtarget OpenholeUD_5013 := [[401.34, -20.7, 180.85], [-0.146245, 0.691818, 0.68943, 0.157118], [0,0,0,0], [9E9, 9E9, 9E9, 9E9, 9E9, 9E9]];
	VAR robtarget OpenholeUD_5014 := [[405.34, -20.7, 180.91], [-0.134962, 0.694107, 0.691843, 0.146126], [0,0,0,0], [9E9, 9E9, 9E9, 9E9, 9E9, 9E9]];
	VAR robtarget OpenholeUD_5015 := [[409.34, -20.7, 180.98], [-0.123331, 0.696268, 0.694142, 0.134783], [0,0,0,0], [9E9, 9E9, 9E9, 9E9, 9E9, 9E9]];
	VAR robtarget OpenholeUD_5016 := [[413.34, -20.7, 181.04], [-0.111366, 0.698282, 0.696309, 0.123102], [0,0,0,0], [9E9, 9E9, 9E9, 9E9, 9E9, 9E9]];
	VAR robtarget OpenholeUD_5017 := [[417.34, -20.7, 181.11], [-0.099084, 0.70013, 0.698325, 0.111098], [0,0,0,0], [9E9, 9E9, 9E9, 9E9, 9E9, 9E9]];
	VAR robtarget OpenholeUD_5018 := [[421.34, -20.7, 181.17], [-0.08651, 0.701795, 0.700172, 0.09879], [0,0,0,0], [9E9, 9E9, 9E9, 9E9, 9E9, 9E9]];
	VAR robtarget OpenholeUD_5019 := [[425.34, -20.7, 181.23], [-0.07367, 0.703259, 0.701833, 0.086204], [0,0,0,0], [9E9, 9E9, 9E9, 9E9, 9E9, 9E9]];
	VAR robtarget OpenholeUD_5020 := [[429.34, -20.7, 181.3], [-0.060595, 0.704506, 0.70329, 0.073367], [0,0,0,0], [9E9, 9E9, 9E9, 9E9, 9E9, 9E9]];
	VAR robtarget OpenholeUD_5021 := [[433.34, -20.7, 181.36], [-0.047321, 0.705522, 0.70453, 0.060311], [0,0,0,0], [9E9, 9E9, 9E9, 9E9, 9E9, 9E9]];
	VAR robtarget OpenholeUD_5022 := [[437.34, -20.7, 181.43], [-0.033887, 0.706294, 0.705538, 0.047073], [0,0,0,0], [9E9, 9E9, 9E9, 9E9, 9E9, 9E9]];
	VAR robtarget OpenholeUD_5023 := [[443.16, -20.7, 181.52], [-0.014122, 0.706966, 0.70657, 0.027547], [0,0,0,0], [9E9, 9E9, 9E9, 9E9, 9E9, 9E9]];
	VAR robtarget OpenholeUD_5024 := [[443.16, -20.7, 181.52], [-0.014122, 0.706966, 0.70657, 0.027547], [0,0,0,0], [9E9, 9E9, 9E9, 9E9, 9E9, 9E9]];
	VAR robtarget OpenholeUD_5025 := [[443.69, -21.9, 181.46], [-0.008236, 0.707059, 0.706477, 0.029827], [0,0,0,0], [9E9, 9E9, 9E9, 9E9, 9E9, 9E9]];
	VAR robtarget OpenholeUD_5026 := [[439.69, -21.9, 181.35], [-0.021848, 0.706769, 0.705782, 0.043256], [0,0,0,0], [9E9, 9E9, 9E9, 9E9, 9E9, 9E9]];
	VAR robtarget OpenholeUD_5027 := [[435.69, -21.9, 181.24], [-0.035375, 0.706221, 0.704841, 0.056559], [0,0,0,0], [9E9, 9E9, 9E9, 9E9, 9E9, 9E9]];
	VAR robtarget OpenholeUD_5028 := [[431.69, -21.9, 181.13], [-0.048772, 0.705423, 0.703664, 0.069695], [0,0,0,0], [9E9, 9E9, 9E9, 9E9, 9E9, 9E9]];
	VAR robtarget OpenholeUD_5029 := [[427.69, -21.9, 181.02], [-0.061999, 0.704384, 0.702263, 0.082626], [0,0,0,0], [9E9, 9E9, 9E9, 9E9, 9E9, 9E9]];
	VAR robtarget OpenholeUD_5030 := [[423.7, -21.9, 180.91], [-0.075018, 0.703116, 0.700653, 0.095319], [0,0,0,0], [9E9, 9E9, 9E9, 9E9, 9E9, 9E9]];
	VAR robtarget OpenholeUD_5031 := [[419.7, -21.9, 180.8], [-0.087795, 0.701635, 0.69885, 0.107744], [0,0,0,0], [9E9, 9E9, 9E9, 9E9, 9E9, 9E9]];
	VAR robtarget OpenholeUD_5032 := [[415.7, -21.9, 180.69], [-0.1003, 0.699957, 0.696872, 0.119875], [0,0,0,0], [9E9, 9E9, 9E9, 9E9, 9E9, 9E9]];
	VAR robtarget OpenholeUD_5033 := [[411.7, -21.9, 180.58], [-0.112507, 0.698099, 0.694736, 0.13169], [0,0,0,0], [9E9, 9E9, 9E9, 9E9, 9E9, 9E9]];
	VAR robtarget OpenholeUD_5034 := [[407.7, -21.9, 180.47], [-0.124394, 0.696079, 0.692461, 0.143172], [0,0,0,0], [9E9, 9E9, 9E9, 9E9, 9E9, 9E9]];
	VAR robtarget OpenholeUD_5035 := [[403.7, -21.9, 180.36], [-0.135944, 0.693916, 0.690065, 0.154307], [0,0,0,0], [9E9, 9E9, 9E9, 9E9, 9E9, 9E9]];
	VAR robtarget OpenholeUD_5036 := [[399.71, -21.9, 180.25], [-0.147143, 0.691628, 0.687566, 0.165085], [0,0,0,0], [9E9, 9E9, 9E9, 9E9, 9E9, 9E9]];
	VAR robtarget OpenholeUD_5037 := [[395.71, -21.9, 180.14], [-0.157983, 0.689233, 0.684982, 0.1755], [0,0,0,0], [9E9, 9E9, 9E9, 9E9, 9E9, 9E9]];
	VAR robtarget OpenholeUD_5038 := [[389.34, -21.9, 179.96], [-0.174484, 0.685241, 0.680731, 0.191326], [0,0,0,0], [9E9, 9E9, 9E9, 9E9, 9E9, 9E9]];
	VAR robtarget OpenholeUD_5039 := [[385.34, -21.9, 179.97], [-0.183051, 0.683002, 0.683002, 0.183051], [0,0,0,0], [9E9, 9E9, 9E9, 9E9, 9E9, 9E9]];
	VAR robtarget OpenholeUD_5040 := [[381.34, -21.9, 179.99], [-0.183051, 0.683002, 0.683002, 0.183051], [0,0,0,0], [9E9, 9E9, 9E9, 9E9, 9E9, 9E9]];
	VAR robtarget OpenholeUD_5041 := [[377.34, -21.9, 180], [-0.183051, 0.683002, 0.683002, 0.183051], [0,0,0,0], [9E9, 9E9, 9E9, 9E9, 9E9, 9E9]];
	VAR robtarget OpenholeUD_5042 := [[373.34, -21.9, 180.01], [-0.183051, 0.683002, 0.683002, 0.183051], [0,0,0,0], [9E9, 9E9, 9E9, 9E9, 9E9, 9E9]];
	VAR robtarget OpenholeUD_5043 := [[369.34, -21.9, 180.02], [-0.183051, 0.683002, 0.683002, 0.183051], [0,0,0,0], [9E9, 9E9, 9E9, 9E9, 9E9, 9E9]];
	VAR robtarget OpenholeUD_5044 := [[369.34, -21.9, 180.02], [-0.183051, 0.683002, 0.683002, 0.183051], [0,0,0,0], [9E9, 9E9, 9E9, 9E9, 9E9, 9E9]];
	VAR robtarget OpenholeUD_5045 := [[369.34, -23.1, 179.33], [-0.183051, 0.683002, 0.683002, 0.183051], [0,0,0,0], [9E9, 9E9, 9E9, 9E9, 9E9, 9E9]];
	VAR robtarget OpenholeUD_5046 := [[373.34, -23.1, 179.32], [-0.183051, 0.683002, 0.683002, 0.183051], [0,0,0,0], [9E9, 9E9, 9E9, 9E9, 9E9, 9E9]];
	VAR robtarget OpenholeUD_5047 := [[377.34, -23.1, 179.31], [-0.183051, 0.683002, 0.683002, 0.183051], [0,0,0,0], [9E9, 9E9, 9E9, 9E9, 9E9, 9E9]];
	VAR robtarget OpenholeUD_5048 := [[381.34, -23.1, 179.29], [-0.183051, 0.683002, 0.683002, 0.183051], [0,0,0,0], [9E9, 9E9, 9E9, 9E9, 9E9, 9E9]];
	VAR robtarget OpenholeUD_5049 := [[385.34, -23.1, 179.28], [-0.183051, 0.683002, 0.683002, 0.183051], [0,0,0,0], [9E9, 9E9, 9E9, 9E9, 9E9, 9E9]];
	VAR robtarget OpenholeUD_5050 := [[389.34, -23.1, 179.27], [-0.17105, 0.686106, 0.679768, 0.19472], [0,0,0,0], [9E9, 9E9, 9E9, 9E9, 9E9, 9E9]];
	VAR robtarget OpenholeUD_5051 := [[393.34, -23.1, 179.43], [-0.160728, 0.688598, 0.682488, 0.184961], [0,0,0,0], [9E9, 9E9, 9E9, 9E9, 9E9, 9E9]];
	VAR robtarget OpenholeUD_5052 := [[397.33, -23.1, 179.58], [-0.15004, 0.691005, 0.685152, 0.174834], [0,0,0,0], [9E9, 9E9, 9E9, 9E9, 9E9, 9E9]];
	VAR robtarget OpenholeUD_5053 := [[401.33, -23.1, 179.74], [-0.138991, 0.693312, 0.687744, 0.164341], [0,0,0,0], [9E9, 9E9, 9E9, 9E9, 9E9, 9E9]];
	VAR robtarget OpenholeUD_5054 := [[405.33, -23.1, 179.9], [-0.127589, 0.695501, 0.690248, 0.153486], [0,0,0,0], [9E9, 9E9, 9E9, 9E9, 9E9, 9E9]];
	VAR robtarget OpenholeUD_5055 := [[409.32, -23.1, 180.05], [-0.115844, 0.697553, 0.692646, 0.142275], [0,0,0,0], [9E9, 9E9, 9E9, 9E9, 9E9, 9E9]];
	VAR robtarget OpenholeUD_5056 := [[413.32, -23.1, 180.21], [-0.103772, 0.699451, 0.694919, 0.130719], [0,0,0,0], [9E9, 9E9, 9E9, 9E9, 9E9, 9E9]];
	VAR robtarget OpenholeUD_5057 := [[417.32, -23.1, 180.37], [-0.091393, 0.701176, 0.69705, 0.118832], [0,0,0,0], [9E9, 9E9, 9E9, 9E9, 9E9, 9E9]];
	VAR robtarget OpenholeUD_5058 := [[421.31, -23.1, 180.52], [-0.078731, 0.70271, 0.69902, 0.106634], [0,0,0,0], [9E9, 9E9, 9E9, 9E9, 9E9, 9E9]];
	VAR robtarget OpenholeUD_5059 := [[425.31, -23.1, 180.68], [-0.065814, 0.704037, 0.700811, 0.094147], [0,0,0,0], [9E9, 9E9, 9E9, 9E9, 9E9, 9E9]];
	VAR robtarget OpenholeUD_5060 := [[429.31, -23.1, 180.84], [-0.052674, 0.705142, 0.702406, 0.081398], [0,0,0,0], [9E9, 9E9, 9E9, 9E9, 9E9, 9E9]];
	VAR robtarget OpenholeUD_5061 := [[433.31, -23.1, 180.99], [-0.039348, 0.706011, 0.703789, 0.068419], [0,0,0,0], [9E9, 9E9, 9E9, 9E9, 9E9, 9E9]];
	VAR robtarget OpenholeUD_5062 := [[437.3, -23.1, 181.15], [-0.025875, 0.706633, 0.704946, 0.055243], [0,0,0,0], [9E9, 9E9, 9E9, 9E9, 9E9, 9E9]];
	VAR robtarget OpenholeUD_5063 := [[444.56, -23.1, 181.43], [-0.001167, 0.707106, 0.70643, 0.030937], [0,0,0,0], [9E9, 9E9, 9E9, 9E9, 9E9, 9E9]];
	VAR robtarget OpenholeUD_5064 := [[444.56, -23.1, 181.43], [-0.001167, 0.707106, 0.70643, 0.030937], [0,0,0,0], [9E9, 9E9, 9E9, 9E9, 9E9, 9E9]];
	VAR robtarget OpenholeUD_5065 := [[446.05, -24.3, 181.45], [0.00799, 0.707062, 0.706471, 0.029979], [0,0,0,0], [9E9, 9E9, 9E9, 9E9, 9E9, 9E9]];
	VAR robtarget OpenholeUD_5066 := [[442.05, -24.3, 181.25], [-0.005655, 0.707084, 0.705772, 0.043429], [0,0,0,0], [9E9, 9E9, 9E9, 9E9, 9E9, 9E9]];
	VAR robtarget OpenholeUD_5067 := [[438.06, -24.3, 181.05], [-0.019255, 0.706845, 0.704825, 0.056762], [0,0,0,0], [9E9, 9E9, 9E9, 9E9, 9E9, 9E9]];
	VAR robtarget OpenholeUD_5068 := [[434.06, -24.3, 180.85], [-0.032766, 0.706347, 0.70364, 0.069938], [0,0,0,0], [9E9, 9E9, 9E9, 9E9, 9E9, 9E9]];
	VAR robtarget OpenholeUD_5069 := [[430.07, -24.3, 180.64], [-0.046146, 0.705599, 0.702228, 0.082919], [0,0,0,0], [9E9, 9E9, 9E9, 9E9, 9E9, 9E9]];
	VAR robtarget OpenholeUD_5070 := [[426.07, -24.3, 180.44], [-0.059352, 0.704611, 0.700605, 0.095669], [0,0,0,0], [9E9, 9E9, 9E9, 9E9, 9E9, 9E9]];
	VAR robtarget OpenholeUD_5071 := [[422.08, -24.3, 180.24], [-0.072349, 0.703396, 0.698786, 0.108157], [0,0,0,0], [9E9, 9E9, 9E9, 9E9, 9E9, 9E9]];
	VAR robtarget OpenholeUD_5072 := [[418.08, -24.3, 180.03], [-0.085103, 0.701967, 0.696789, 0.120357], [0,0,0,0], [9E9, 9E9, 9E9, 9E9, 9E9, 9E9]];
	VAR robtarget OpenholeUD_5073 := [[414.09, -24.3, 179.83], [-0.097584, 0.700341, 0.69463, 0.132245], [0,0,0,0], [9E9, 9E9, 9E9, 9E9, 9E9, 9E9]];
	VAR robtarget OpenholeUD_5074 := [[410.09, -24.3, 179.63], [-0.109766, 0.698535, 0.69233, 0.143802], [0,0,0,0], [9E9, 9E9, 9E9, 9E9, 9E9, 9E9]];
	VAR robtarget OpenholeUD_5075 := [[406.1, -24.3, 179.43], [-0.121629, 0.696568, 0.689906, 0.155014], [0,0,0,0], [9E9, 9E9, 9E9, 9E9, 9E9, 9E9]];
	VAR robtarget OpenholeUD_5076 := [[402.1, -24.3, 179.22], [-0.133156, 0.694456, 0.687377, 0.165869], [0,0,0,0], [9E9, 9E9, 9E9, 9E9, 9E9, 9E9]];
	VAR robtarget OpenholeUD_5077 := [[398.11, -24.3, 179.02], [-0.144334, 0.692219, 0.68476, 0.176361], [0,0,0,0], [9E9, 9E9, 9E9, 9E9, 9E9, 9E9]];
	VAR robtarget OpenholeUD_5078 := [[394.11, -24.3, 178.82], [-0.155155, 0.689875, 0.682073, 0.186486], [0,0,0,0], [9E9, 9E9, 9E9, 9E9, 9E9, 9E9]];
	VAR robtarget OpenholeUD_5079 := [[389.34, -24.3, 178.58], [-0.167613, 0.686954, 0.678788, 0.198107], [0,0,0,0], [9E9, 9E9, 9E9, 9E9, 9E9, 9E9]];
	VAR robtarget OpenholeUD_5080 := [[385.34, -24.3, 178.59], [-0.183051, 0.683002, 0.683002, 0.183051], [0,0,0,0], [9E9, 9E9, 9E9, 9E9, 9E9, 9E9]];
	VAR robtarget OpenholeUD_5081 := [[381.34, -24.3, 178.6], [-0.183051, 0.683002, 0.683002, 0.183051], [0,0,0,0], [9E9, 9E9, 9E9, 9E9, 9E9, 9E9]];
	VAR robtarget OpenholeUD_5082 := [[377.34, -24.3, 178.61], [-0.183051, 0.683002, 0.683002, 0.183051], [0,0,0,0], [9E9, 9E9, 9E9, 9E9, 9E9, 9E9]];
	VAR robtarget OpenholeUD_5083 := [[369.34, -24.3, 178.64], [-0.183051, 0.683002, 0.683002, 0.183051], [0,0,0,0], [9E9, 9E9, 9E9, 9E9, 9E9, 9E9]];
	VAR robtarget OpenholeUD_5084 := [[369.34, -24.3, 178.64], [-0.183051, 0.683002, 0.683002, 0.183051], [0,0,0,0], [9E9, 9E9, 9E9, 9E9, 9E9, 9E9]];
	VAR robtarget OpenholeUD_5085 := [[369.34, -25.5, 177.95], [-0.183051, 0.683002, 0.683002, 0.183051], [0,0,0,0], [9E9, 9E9, 9E9, 9E9, 9E9, 9E9]];
	VAR robtarget OpenholeUD_5086 := [[373.34, -25.5, 177.93], [-0.183051, 0.683002, 0.683002, 0.183051], [0,0,0,0], [9E9, 9E9, 9E9, 9E9, 9E9, 9E9]];
	VAR robtarget OpenholeUD_5087 := [[377.34, -25.5, 177.92], [-0.183051, 0.683002, 0.683002, 0.183051], [0,0,0,0], [9E9, 9E9, 9E9, 9E9, 9E9, 9E9]];
	VAR robtarget OpenholeUD_5088 := [[381.34, -25.5, 177.91], [-0.183051, 0.683002, 0.683002, 0.183051], [0,0,0,0], [9E9, 9E9, 9E9, 9E9, 9E9, 9E9]];
	VAR robtarget OpenholeUD_5089 := [[385.34, -25.5, 177.9], [-0.183051, 0.683002, 0.683002, 0.183051], [0,0,0,0], [9E9, 9E9, 9E9, 9E9, 9E9, 9E9]];
	VAR robtarget OpenholeUD_5090 := [[389.34, -25.5, 177.88], [-0.164176, 0.687784, 0.677793, 0.201487], [0,0,0,0], [9E9, 9E9, 9E9, 9E9, 9E9, 9E9]];
	VAR robtarget OpenholeUD_5091 := [[393.33, -25.5, 178.13], [-0.153728, 0.690194, 0.680576, 0.191877], [0,0,0,0], [9E9, 9E9, 9E9, 9E9, 9E9, 9E9]];
	VAR robtarget OpenholeUD_5092 := [[397.32, -25.5, 178.38], [-0.142918, 0.692513, 0.68331, 0.1819], [0,0,0,0], [9E9, 9E9, 9E9, 9E9, 9E9, 9E9]];
	VAR robtarget OpenholeUD_5093 := [[401.31, -25.5, 178.63], [-0.131752, 0.694724, 0.685981, 0.171553], [0,0,0,0], [9E9, 9E9, 9E9, 9E9, 9E9, 9E9]];
	VAR robtarget OpenholeUD_5094 := [[405.3, -25.5, 178.88], [-0.120237, 0.696809, 0.688571, 0.16084], [0,0,0,0], [9E9, 9E9, 9E9, 9E9, 9E9, 9E9]];
	VAR robtarget OpenholeUD_5095 := [[409.3, -25.5, 179.13], [-0.108387, 0.69875, 0.691064, 0.149767], [0,0,0,0], [9E9, 9E9, 9E9, 9E9, 9E9, 9E9]];
	VAR robtarget OpenholeUD_5096 := [[413.29, -25.5, 179.38], [-0.096218, 0.70053, 0.693441, 0.138344], [0,0,0,0], [9E9, 9E9, 9E9, 9E9, 9E9, 9E9]];
	VAR robtarget OpenholeUD_5097 := [[417.28, -25.5, 179.62], [-0.083751, 0.702129, 0.695684, 0.126583], [0,0,0,0], [9E9, 9E9, 9E9, 9E9, 9E9, 9E9]];
	VAR robtarget OpenholeUD_5098 := [[421.27, -25.5, 179.87], [-0.071011, 0.703532, 0.697774, 0.114502], [0,0,0,0], [9E9, 9E9, 9E9, 9E9, 9E9, 9E9]];
	VAR robtarget OpenholeUD_5099 := [[425.27, -25.5, 180.12], [-0.058027, 0.704722, 0.699693, 0.102123], [0,0,0,0], [9E9, 9E9, 9E9, 9E9, 9E9, 9E9]];
	VAR robtarget OpenholeUD_5100 := [[429.26, -25.5, 180.37], [-0.044832, 0.705684, 0.701423, 0.089472], [0,0,0,0], [9E9, 9E9, 9E9, 9E9, 9E9, 9E9]];
	VAR robtarget OpenholeUD_5101 := [[433.25, -25.5, 180.62], [-0.031463, 0.706406, 0.702948, 0.076578], [0,0,0,0], [9E9, 9E9, 9E9, 9E9, 9E9, 9E9]];
	VAR robtarget OpenholeUD_5102 := [[437.24, -25.5, 180.87], [-0.017962, 0.706879, 0.704252, 0.063475], [0,0,0,0], [9E9, 9E9, 9E9, 9E9, 9E9, 9E9]];
	VAR robtarget OpenholeUD_5103 := [[441.23, -25.5, 181.12], [-0.004369, 0.707093, 0.705323, 0.0502], [0,0,0,0], [9E9, 9E9, 9E9, 9E9, 9E9, 9E9]];
	VAR robtarget OpenholeUD_5104 := [[445.23, -25.5, 181.36], [0.00927, 0.707046, 0.706149, 0.036793], [0,0,0,0], [9E9, 9E9, 9E9, 9E9, 9E9, 9E9]];
	VAR robtarget OpenholeUD_5105 := [[449.22, -25.5, 181.61], [0.022909, 0.706736, 0.706723, 0.023296], [0,0,0,0], [9E9, 9E9, 9E9, 9E9, 9E9, 9E9]];
	VAR robtarget OpenholeUD_5106 := [[453.21, -25.5, 181.86], [0.036502, 0.706164, 0.70704, 0.009753], [0,0,0,0], [9E9, 9E9, 9E9, 9E9, 9E9, 9E9]];
	VAR robtarget OpenholeUD_5107 := [[457.2, -25.5, 182.11], [0.050006, 0.705336, 0.707097, -0.003791], [0,0,0,0], [9E9, 9E9, 9E9, 9E9, 9E9, 9E9]];
	VAR robtarget OpenholeUD_5108 := [[461.2, -25.5, 182.36], [0.063375, 0.704261, 0.706895, -0.017293], [0,0,0,0], [9E9, 9E9, 9E9, 9E9, 9E9, 9E9]];
	VAR robtarget OpenholeUD_5109 := [[465.19, -25.5, 182.61], [0.076569, 0.702949, 0.70644, -0.030708], [0,0,0,0], [9E9, 9E9, 9E9, 9E9, 9E9, 9E9]];
	VAR robtarget OpenholeUD_5110 := [[469.18, -25.5, 182.86], [0.089549, 0.701414, 0.705737, -0.043996], [0,0,0,0], [9E9, 9E9, 9E9, 9E9, 9E9, 9E9]];
	VAR robtarget OpenholeUD_5111 := [[473.17, -25.5, 183.11], [0.102282, 0.69967, 0.704796, -0.057117], [0,0,0,0], [9E9, 9E9, 9E9, 9E9, 9E9, 9E9]];
	VAR robtarget OpenholeUD_5112 := [[477.16, -25.5, 183.35], [0.114736, 0.697736, 0.70363, -0.070034], [0,0,0,0], [9E9, 9E9, 9E9, 9E9, 9E9, 9E9]];
	VAR robtarget OpenholeUD_5113 := [[481.16, -25.5, 183.6], [0.126886, 0.695629, 0.702252, -0.082715], [0,0,0,0], [9E9, 9E9, 9E9, 9E9, 9E9, 9E9]];
	VAR robtarget OpenholeUD_5114 := [[485.15, -25.5, 183.85], [0.138709, 0.693369, 0.700678, -0.09513], [0,0,0,0], [9E9, 9E9, 9E9, 9E9, 9E9, 9E9]];
	VAR robtarget OpenholeUD_5115 := [[489.14, -25.5, 184.1], [0.150187, 0.690973, 0.698925, -0.107256], [0,0,0,0], [9E9, 9E9, 9E9, 9E9, 9E9, 9E9]];
	VAR robtarget OpenholeUD_5116 := [[493.13, -25.5, 184.35], [0.161308, 0.688462, 0.697009, -0.119071], [0,0,0,0], [9E9, 9E9, 9E9, 9E9, 9E9, 9E9]];
	VAR robtarget OpenholeUD_5117 := [[497.13, -25.5, 184.6], [0.172062, 0.685853, 0.694949, -0.130558], [0,0,0,0], [9E9, 9E9, 9E9, 9E9, 9E9, 9E9]];
	VAR robtarget OpenholeUD_5118 := [[501.12, -25.5, 184.85], [0.182444, 0.683165, 0.692763, -0.141704], [0,0,0,0], [9E9, 9E9, 9E9, 9E9, 9E9, 9E9]];
	VAR robtarget OpenholeUD_5119 := [[505.11, -25.5, 185.1], [0.192451, 0.680414, 0.690466, -0.1525], [0,0,0,0], [9E9, 9E9, 9E9, 9E9, 9E9, 9E9]];
	VAR robtarget OpenholeUD_5120 := [[509.36, -25.5, 185.36], [0.183051, 0.683002, 0.683002, -0.183051], [0,0,0,0], [9E9, 9E9, 9E9, 9E9, 9E9, 9E9]];
	VAR robtarget OpenholeUD_5121 := [[513.36, -25.5, 185.35], [0.183051, 0.683002, 0.683002, -0.183051], [0,0,0,0], [9E9, 9E9, 9E9, 9E9, 9E9, 9E9]];
	VAR robtarget OpenholeUD_5122 := [[517.36, -25.5, 185.33], [0.183051, 0.683002, 0.683002, -0.183051], [0,0,0,0], [9E9, 9E9, 9E9, 9E9, 9E9, 9E9]];
	VAR robtarget OpenholeUD_5123 := [[521.36, -25.5, 185.32], [0.183051, 0.683002, 0.683002, -0.183051], [0,0,0,0], [9E9, 9E9, 9E9, 9E9, 9E9, 9E9]];
	VAR robtarget OpenholeUD_5124 := [[529.36, -25.5, 185.3], [0.183051, 0.683002, 0.683002, -0.183051], [0,0,0,0], [9E9, 9E9, 9E9, 9E9, 9E9, 9E9]];
	VAR robtarget OpenholeUD_5125 := [[529.36, -25.5, 185.3], [0.183051, 0.683002, 0.683002, -0.183051], [0,0,0,0], [9E9, 9E9, 9E9, 9E9, 9E9, 9E9]];
	VAR robtarget OpenholeUD_5126 := [[529.36, -26.7, 185.99], [0.183051, 0.683002, 0.683002, -0.183051], [0,0,0,0], [9E9, 9E9, 9E9, 9E9, 9E9, 9E9]];
	VAR robtarget OpenholeUD_5127 := [[525.36, -26.7, 186], [0.183051, 0.683002, 0.683002, -0.183051], [0,0,0,0], [9E9, 9E9, 9E9, 9E9, 9E9, 9E9]];
	VAR robtarget OpenholeUD_5128 := [[521.36, -26.7, 186.02], [0.183051, 0.683002, 0.683002, -0.183051], [0,0,0,0], [9E9, 9E9, 9E9, 9E9, 9E9, 9E9]];
	VAR robtarget OpenholeUD_5129 := [[517.36, -26.7, 186.03], [0.183051, 0.683002, 0.683002, -0.183051], [0,0,0,0], [9E9, 9E9, 9E9, 9E9, 9E9, 9E9]];
	VAR robtarget OpenholeUD_5130 := [[509.36, -26.7, 186.05], [0.183051, 0.683002, 0.683002, -0.183051], [0,0,0,0], [9E9, 9E9, 9E9, 9E9, 9E9, 9E9]];
	VAR robtarget OpenholeUD_5131 := [[505.37, -26.7, 185.76], [0.196536, 0.679245, 0.691078, -0.149705], [0,0,0,0], [9E9, 9E9, 9E9, 9E9, 9E9, 9E9]];
	VAR robtarget OpenholeUD_5132 := [[501.38, -26.7, 185.46], [0.186631, 0.682033, 0.693335, -0.138874], [0,0,0,0], [9E9, 9E9, 9E9, 9E9, 9E9, 9E9]];
	VAR robtarget OpenholeUD_5133 := [[497.39, -26.7, 185.17], [0.17635, 0.684763, 0.695481, -0.127696], [0,0,0,0], [9E9, 9E9, 9E9, 9E9, 9E9, 9E9]];
	VAR robtarget OpenholeUD_5134 := [[493.4, -26.7, 184.87], [0.165695, 0.687419, 0.697497, -0.116179], [0,0,0,0], [9E9, 9E9, 9E9, 9E9, 9E9, 9E9]];
	VAR robtarget OpenholeUD_5135 := [[489.42, -26.7, 184.58], [0.15467, 0.689983, 0.699367, -0.104336], [0,0,0,0], [9E9, 9E9, 9E9, 9E9, 9E9, 9E9]];
	VAR robtarget OpenholeUD_5136 := [[485.43, -26.7, 184.29], [0.143285, 0.692437, 0.701072, -0.092186], [0,0,0,0], [9E9, 9E9, 9E9, 9E9, 9E9, 9E9]];
	VAR robtarget OpenholeUD_5137 := [[481.44, -26.7, 183.99], [0.131551, 0.694762, 0.702595, -0.079748], [0,0,0,0], [9E9, 9E9, 9E9, 9E9, 9E9, 9E9]];
	VAR robtarget OpenholeUD_5138 := [[477.45, -26.7, 183.7], [0.119485, 0.696939, 0.703921, -0.067049], [0,0,0,0], [9E9, 9E9, 9E9, 9E9, 9E9, 9E9]];
	VAR robtarget OpenholeUD_5139 := [[473.46, -26.7, 183.4], [0.107108, 0.698948, 0.705033, -0.054116], [0,0,0,0], [9E9, 9E9, 9E9, 9E9, 9E9, 9E9]];
	VAR robtarget OpenholeUD_5140 := [[469.47, -26.7, 183.11], [0.094446, 0.700771, 0.705918, -0.040984], [0,0,0,0], [9E9, 9E9, 9E9, 9E9, 9E9, 9E9]];
	VAR robtarget OpenholeUD_5141 := [[465.48, -26.7, 182.81], [0.081528, 0.702391, 0.706564, -0.027689], [0,0,0,0], [9E9, 9E9, 9E9, 9E9, 9E9, 9E9]];
	VAR robtarget OpenholeUD_5142 := [[461.49, -26.7, 182.52], [0.068388, 0.703792, 0.706963, -0.014269], [0,0,0,0], [9E9, 9E9, 9E9, 9E9, 9E9, 9E9]];
	VAR robtarget OpenholeUD_5143 := [[457.5, -26.7, 182.22], [0.055063, 0.70496, 0.707106, -0.000768], [0,0,0,0], [9E9, 9E9, 9E9, 9E9, 9E9, 9E9]];
	VAR robtarget OpenholeUD_5144 := [[453.51, -26.7, 181.93], [0.041595, 0.705882, 0.706991, 0.012773], [0,0,0,0], [9E9, 9E9, 9E9, 9E9, 9E9, 9E9]];
	VAR robtarget OpenholeUD_5145 := [[449.52, -26.7, 181.63], [0.028025, 0.706551, 0.706617, 0.026308], [0,0,0,0], [9E9, 9E9, 9E9, 9E9, 9E9, 9E9]];
	VAR robtarget OpenholeUD_5146 := [[445.54, -26.7, 181.34], [0.014398, 0.70696, 0.705986, 0.039793], [0,0,0,0], [9E9, 9E9, 9E9, 9E9, 9E9, 9E9]];
	VAR robtarget OpenholeUD_5147 := [[441.55, -26.7, 181.05], [0.000761, 0.707106, 0.705104, 0.053185], [0,0,0,0], [9E9, 9E9, 9E9, 9E9, 9E9, 9E9]];
	VAR robtarget OpenholeUD_5148 := [[437.56, -26.7, 180.75], [-0.01284, 0.70699, 0.703978, 0.066441], [0,0,0,0], [9E9, 9E9, 9E9, 9E9, 9E9, 9E9]];
	VAR robtarget OpenholeUD_5149 := [[433.57, -26.7, 180.46], [-0.026362, 0.706615, 0.702621, 0.079522], [0,0,0,0], [9E9, 9E9, 9E9, 9E9, 9E9, 9E9]];
	VAR robtarget OpenholeUD_5150 := [[429.58, -26.7, 180.16], [-0.039761, 0.705988, 0.701045, 0.09239], [0,0,0,0], [9E9, 9E9, 9E9, 9E9, 9E9, 9E9]];
	VAR robtarget OpenholeUD_5151 := [[425.59, -26.7, 179.87], [-0.052996, 0.705118, 0.699266, 0.105013], [0,0,0,0], [9E9, 9E9, 9E9, 9E9, 9E9, 9E9]];
	VAR robtarget OpenholeUD_5152 := [[421.6, -26.7, 179.57], [-0.06603, 0.704017, 0.697299, 0.11736], [0,0,0,0], [9E9, 9E9, 9E9, 9E9, 9E9, 9E9]];
	VAR robtarget OpenholeUD_5153 := [[417.61, -26.7, 179.28], [-0.078828, 0.702699, 0.695165, 0.129407], [0,0,0,0], [9E9, 9E9, 9E9, 9E9, 9E9, 9E9]];
	VAR robtarget OpenholeUD_5154 := [[413.62, -26.7, 178.98], [-0.09136, 0.70118, 0.692879, 0.141132], [0,0,0,0], [9E9, 9E9, 9E9, 9E9, 9E9, 9E9]];
	VAR robtarget OpenholeUD_5155 := [[409.63, -26.7, 178.69], [-0.103601, 0.699476, 0.690463, 0.152517], [0,0,0,0], [9E9, 9E9, 9E9, 9E9, 9E9, 9E9]];
	VAR robtarget OpenholeUD_5156 := [[405.64, -26.7, 178.39], [-0.115529, 0.697605, 0.687933, 0.16355], [0,0,0,0], [9E9, 9E9, 9E9, 9E9, 9E9, 9E9]];
	VAR robtarget OpenholeUD_5157 := [[401.65, -26.7, 178.1], [-0.127126, 0.695585, 0.685308, 0.174222], [0,0,0,0], [9E9, 9E9, 9E9, 9E9, 9E9, 9E9]];
	VAR robtarget OpenholeUD_5158 := [[397.67, -26.7, 177.81], [-0.13838, 0.693434, 0.682605, 0.184526], [0,0,0,0], [9E9, 9E9, 9E9, 9E9, 9E9, 9E9]];
	VAR robtarget OpenholeUD_5159 := [[393.68, -26.7, 177.51], [-0.149279, 0.69117, 0.679842, 0.194461], [0,0,0,0], [9E9, 9E9, 9E9, 9E9, 9E9, 9E9]];
	VAR robtarget OpenholeUD_5160 := [[389.33, -26.7, 177.19], [-0.160738, 0.688595, 0.676782, 0.204858], [0,0,0,0], [9E9, 9E9, 9E9, 9E9, 9E9, 9E9]];
	VAR robtarget OpenholeUD_5161 := [[385.33, -26.7, 177.2], [-0.183051, 0.683002, 0.683002, 0.183051], [0,0,0,0], [9E9, 9E9, 9E9, 9E9, 9E9, 9E9]];
	VAR robtarget OpenholeUD_5162 := [[381.33, -26.7, 177.22], [-0.183051, 0.683002, 0.683002, 0.183051], [0,0,0,0], [9E9, 9E9, 9E9, 9E9, 9E9, 9E9]];
	VAR robtarget OpenholeUD_5163 := [[377.33, -26.7, 177.23], [-0.183051, 0.683002, 0.683002, 0.183051], [0,0,0,0], [9E9, 9E9, 9E9, 9E9, 9E9, 9E9]];
	VAR robtarget OpenholeUD_5164 := [[373.33, -26.7, 177.24], [-0.183051, 0.683002, 0.683002, 0.183051], [0,0,0,0], [9E9, 9E9, 9E9, 9E9, 9E9, 9E9]];
	VAR robtarget OpenholeUD_5165 := [[369.33, -26.7, 177.25], [-0.183051, 0.683002, 0.683002, 0.183051], [0,0,0,0], [9E9, 9E9, 9E9, 9E9, 9E9, 9E9]];
	VAR robtarget OpenholeUD_5166 := [[369.33, -26.7, 177.25], [-0.183051, 0.683002, 0.683002, 0.183051], [0,0,0,0], [9E9, 9E9, 9E9, 9E9, 9E9, 9E9]];
	VAR robtarget OpenholeUD_5167 := [[369.33, -27.9, 176.56], [-0.183051, 0.683002, 0.683002, 0.183051], [0,0,0,0], [9E9, 9E9, 9E9, 9E9, 9E9, 9E9]];
	VAR robtarget OpenholeUD_5168 := [[373.33, -27.9, 176.55], [-0.183051, 0.683002, 0.683002, 0.183051], [0,0,0,0], [9E9, 9E9, 9E9, 9E9, 9E9, 9E9]];
	VAR robtarget OpenholeUD_5169 := [[377.33, -27.9, 176.53], [-0.183051, 0.683002, 0.683002, 0.183051], [0,0,0,0], [9E9, 9E9, 9E9, 9E9, 9E9, 9E9]];
	VAR robtarget OpenholeUD_5170 := [[381.33, -27.9, 176.52], [-0.183051, 0.683002, 0.683002, 0.183051], [0,0,0,0], [9E9, 9E9, 9E9, 9E9, 9E9, 9E9]];
	VAR robtarget OpenholeUD_5171 := [[385.33, -27.9, 176.51], [-0.183051, 0.683002, 0.683002, 0.183051], [0,0,0,0], [9E9, 9E9, 9E9, 9E9, 9E9, 9E9]];
	VAR robtarget OpenholeUD_5172 := [[389.33, -27.9, 176.5], [-0.1573, 0.689389, 0.675755, 0.208219], [0,0,0,0], [9E9, 9E9, 9E9, 9E9, 9E9, 9E9]];
	VAR robtarget OpenholeUD_5173 := [[393.32, -27.9, 176.84], [-0.146734, 0.691715, 0.678596, 0.198764], [0,0,0,0], [9E9, 9E9, 9E9, 9E9, 9E9, 9E9]];
	VAR robtarget OpenholeUD_5174 := [[397.3, -27.9, 177.18], [-0.13581, 0.693942, 0.681397, 0.18894], [0,0,0,0], [9E9, 9E9, 9E9, 9E9, 9E9, 9E9]];
	VAR robtarget OpenholeUD_5175 := [[401.29, -27.9, 177.52], [-0.124534, 0.696054, 0.684142, 0.178745], [0,0,0,0], [9E9, 9E9, 9E9, 9E9, 9E9, 9E9]];
	VAR robtarget OpenholeUD_5176 := [[405.27, -27.9, 177.86], [-0.112916, 0.698033, 0.686815, 0.168181], [0,0,0,0], [9E9, 9E9, 9E9, 9E9, 9E9, 9E9]];
	VAR robtarget OpenholeUD_5177 := [[409.26, -27.9, 178.2], [-0.10097, 0.699861, 0.6894, 0.157252], [0,0,0,0], [9E9, 9E9, 9E9, 9E9, 9E9, 9E9]];
	VAR robtarget OpenholeUD_5178 := [[413.24, -27.9, 178.54], [-0.088714, 0.70152, 0.691877, 0.145968], [0,0,0,0], [9E9, 9E9, 9E9, 9E9, 9E9, 9E9]];
	VAR robtarget OpenholeUD_5179 := [[417.23, -27.9, 178.88], [-0.076168, 0.702992, 0.694228, 0.134341], [0,0,0,0], [9E9, 9E9, 9E9, 9E9, 9E9, 9E9]];
	VAR robtarget OpenholeUD_5180 := [[421.21, -27.9, 179.22], [-0.06336, 0.704262, 0.696435, 0.122385], [0,0,0,0], [9E9, 9E9, 9E9, 9E9, 9E9, 9E9]];
	VAR robtarget OpenholeUD_5181 := [[425.2, -27.9, 179.56], [-0.050318, 0.705314, 0.698479, 0.110123], [0,0,0,0], [9E9, 9E9, 9E9, 9E9, 9E9, 9E9]];
	VAR robtarget OpenholeUD_5182 := [[429.19, -27.9, 179.9], [-0.037079, 0.706134, 0.700342, 0.097577], [0,0,0,0], [9E9, 9E9, 9E9, 9E9, 9E9, 9E9]];
	VAR robtarget OpenholeUD_5183 := [[433.17, -27.9, 180.24], [-0.023678, 0.70671, 0.702006, 0.084778], [0,0,0,0], [9E9, 9E9, 9E9, 9E9, 9E9, 9E9]];
	VAR robtarget OpenholeUD_5184 := [[437.16, -27.9, 180.58], [-0.010157, 0.707034, 0.703456, 0.071757], [0,0,0,0], [9E9, 9E9, 9E9, 9E9, 9E9, 9E9]];
	VAR robtarget OpenholeUD_5185 := [[441.14, -27.9, 180.92], [0.003441, 0.707098, 0.704679, 0.05855], [0,0,0,0], [9E9, 9E9, 9E9, 9E9, 9E9, 9E9]];
	VAR robtarget OpenholeUD_5186 := [[445.13, -27.9, 181.26], [0.017072, 0.706901, 0.705661, 0.045197], [0,0,0,0], [9E9, 9E9, 9E9, 9E9, 9E9, 9E9]];
	VAR robtarget OpenholeUD_5187 := [[449.11, -27.9, 181.6], [0.030689, 0.706441, 0.706394, 0.031739], [0,0,0,0], [9E9, 9E9, 9E9, 9E9, 9E9, 9E9]];
	VAR robtarget OpenholeUD_5188 := [[453.1, -27.9, 181.94], [0.044247, 0.705721, 0.706872, 0.018219], [0,0,0,0], [9E9, 9E9, 9E9, 9E9, 9E9, 9E9]];
	VAR robtarget OpenholeUD_5189 := [[457.08, -27.9, 182.28], [0.057701, 0.704749, 0.707091, 0.004682], [0,0,0,0], [9E9, 9E9, 9E9, 9E9, 9E9, 9E9]];
	VAR robtarget OpenholeUD_5190 := [[461.07, -27.9, 182.62], [0.071009, 0.703532, 0.707052, -0.008828], [0,0,0,0], [9E9, 9E9, 9E9, 9E9, 9E9, 9E9]];
	VAR robtarget OpenholeUD_5191 := [[465.06, -27.9, 182.96], [0.08413, 0.702084, 0.706756, -0.022267], [0,0,0,0], [9E9, 9E9, 9E9, 9E9, 9E9, 9E9]];
	VAR robtarget OpenholeUD_5192 := [[469.04, -27.9, 183.3], [0.097026, 0.700418, 0.70621, -0.035593], [0,0,0,0], [9E9, 9E9, 9E9, 9E9, 9E9, 9E9]];
	VAR robtarget OpenholeUD_5193 := [[473.03, -27.9, 183.64], [0.109665, 0.698551, 0.705423, -0.048767], [0,0,0,0], [9E9, 9E9, 9E9, 9E9, 9E9, 9E9]];
	VAR robtarget OpenholeUD_5194 := [[477.01, -27.9, 183.98], [0.122016, 0.6965, 0.704405, -0.061751], [0,0,0,0], [9E9, 9E9, 9E9, 9E9, 9E9, 9E9]];
	VAR robtarget OpenholeUD_5195 := [[481, -27.9, 184.32], [0.134055, 0.694283, 0.70317, -0.074511], [0,0,0,0], [9E9, 9E9, 9E9, 9E9, 9E9, 9E9]];
	VAR robtarget OpenholeUD_5196 := [[484.98, -27.9, 184.66], [0.14576, 0.691921, 0.701732, -0.087017], [0,0,0,0], [9E9, 9E9, 9E9, 9E9, 9E9, 9E9]];
	VAR robtarget OpenholeUD_5197 := [[488.97, -27.9, 185], [0.157115, 0.689431, 0.700108, -0.099244], [0,0,0,0], [9E9, 9E9, 9E9, 9E9, 9E9, 9E9]];
	VAR robtarget OpenholeUD_5198 := [[492.95, -27.9, 185.34], [0.168108, 0.686833, 0.698313, -0.111169], [0,0,0,0], [9E9, 9E9, 9E9, 9E9, 9E9, 9E9]];
	VAR robtarget OpenholeUD_5199 := [[496.94, -27.9, 185.69], [0.178731, 0.684146, 0.696367, -0.122774], [0,0,0,0], [9E9, 9E9, 9E9, 9E9, 9E9, 9E9]];
	VAR robtarget OpenholeUD_5200 := [[500.92, -27.9, 186.03], [0.188979, 0.681386, 0.694285, -0.134045], [0,0,0,0], [9E9, 9E9, 9E9, 9E9, 9E9, 9E9]];
	VAR robtarget OpenholeUD_5201 := [[504.91, -27.9, 186.37], [0.19885, 0.678571, 0.692086, -0.144972], [0,0,0,0], [9E9, 9E9, 9E9, 9E9, 9E9, 9E9]];
	VAR robtarget OpenholeUD_5202 := [[509.36, -27.9, 186.75], [0.183051, 0.683002, 0.683002, -0.183051], [0,0,0,0], [9E9, 9E9, 9E9, 9E9, 9E9, 9E9]];
	VAR robtarget OpenholeUD_5203 := [[513.36, -27.9, 186.73], [0.183051, 0.683002, 0.683002, -0.183051], [0,0,0,0], [9E9, 9E9, 9E9, 9E9, 9E9, 9E9]];
	VAR robtarget OpenholeUD_5204 := [[517.36, -27.9, 186.72], [0.183051, 0.683002, 0.683002, -0.183051], [0,0,0,0], [9E9, 9E9, 9E9, 9E9, 9E9, 9E9]];
	VAR robtarget OpenholeUD_5205 := [[521.36, -27.9, 186.71], [0.183051, 0.683002, 0.683002, -0.183051], [0,0,0,0], [9E9, 9E9, 9E9, 9E9, 9E9, 9E9]];
	VAR robtarget OpenholeUD_5206 := [[525.36, -27.9, 186.7], [0.183051, 0.683002, 0.683002, -0.183051], [0,0,0,0], [9E9, 9E9, 9E9, 9E9, 9E9, 9E9]];
	VAR robtarget OpenholeUD_5207 := [[529.36, -27.9, 186.68], [0.183051, 0.683002, 0.683002, -0.183051], [0,0,0,0], [9E9, 9E9, 9E9, 9E9, 9E9, 9E9]];
	VAR robtarget OpenholeUD_5208 := [[529.36, -27.9, 186.68], [0.183051, 0.683002, 0.683002, -0.183051], [0,0,0,0], [9E9, 9E9, 9E9, 9E9, 9E9, 9E9]];
	VAR robtarget OpenholeUD_5209 := [[529.37, -29.1, 187.38], [0.183051, 0.683002, 0.683002, -0.183051], [0,0,0,0], [9E9, 9E9, 9E9, 9E9, 9E9, 9E9]];
	VAR robtarget OpenholeUD_5210 := [[525.37, -29.1, 187.39], [0.183051, 0.683002, 0.683002, -0.183051], [0,0,0,0], [9E9, 9E9, 9E9, 9E9, 9E9, 9E9]];
	VAR robtarget OpenholeUD_5211 := [[521.37, -29.1, 187.4], [0.183051, 0.683002, 0.683002, -0.183051], [0,0,0,0], [9E9, 9E9, 9E9, 9E9, 9E9, 9E9]];
	VAR robtarget OpenholeUD_5212 := [[517.37, -29.1, 187.41], [0.183051, 0.683002, 0.683002, -0.183051], [0,0,0,0], [9E9, 9E9, 9E9, 9E9, 9E9, 9E9]];
	VAR robtarget OpenholeUD_5213 := [[513.37, -29.1, 187.43], [0.183051, 0.683002, 0.683002, -0.183051], [0,0,0,0], [9E9, 9E9, 9E9, 9E9, 9E9, 9E9]];
	VAR robtarget OpenholeUD_5214 := [[509.37, -29.1, 187.44], [0.183051, 0.683002, 0.683002, -0.183051], [0,0,0,0], [9E9, 9E9, 9E9, 9E9, 9E9, 9E9]];
	VAR robtarget OpenholeUD_5215 := [[505.38, -29.1, 187.05], [0.203421, 0.677215, 0.692545, -0.142761], [0,0,0,0], [9E9, 9E9, 9E9, 9E9, 9E9, 9E9]];
	VAR robtarget OpenholeUD_5216 := [[501.4, -29.1, 186.67], [0.193674, 0.680066, 0.694711, -0.131823], [0,0,0,0], [9E9, 9E9, 9E9, 9E9, 9E9, 9E9]];
	VAR robtarget OpenholeUD_5217 := [[497.42, -29.1, 186.28], [0.183549, 0.682869, 0.696757, -0.120541], [0,0,0,0], [9E9, 9E9, 9E9, 9E9, 9E9, 9E9]];
	VAR robtarget OpenholeUD_5218 := [[493.44, -29.1, 185.9], [0.173048, 0.685605, 0.698666, -0.108928], [0,0,0,0], [9E9, 9E9, 9E9, 9E9, 9E9, 9E9]];
	VAR robtarget OpenholeUD_5219 := [[489.46, -29.1, 185.51], [0.162174, 0.688258, 0.700423, -0.096996], [0,0,0,0], [9E9, 9E9, 9E9, 9E9, 9E9, 9E9]];
	VAR robtarget OpenholeUD_5220 := [[485.48, -29.1, 185.12], [0.150935, 0.69081, 0.702008, -0.084764], [0,0,0,0], [9E9, 9E9, 9E9, 9E9, 9E9, 9E9]];
	VAR robtarget OpenholeUD_5221 := [[481.5, -29.1, 184.74], [0.139341, 0.693242, 0.703406, -0.072254], [0,0,0,0], [9E9, 9E9, 9E9, 9E9, 9E9, 9E9]];
	VAR robtarget OpenholeUD_5222 := [[477.52, -29.1, 184.35], [0.127407, 0.695534, 0.7046, -0.059492], [0,0,0,0], [9E9, 9E9, 9E9, 9E9, 9E9, 9E9]];
	VAR robtarget OpenholeUD_5223 := [[473.53, -29.1, 183.97], [0.115155, 0.697667, 0.705576, -0.046509], [0,0,0,0], [9E9, 9E9, 9E9, 9E9, 9E9, 9E9]];
	VAR robtarget OpenholeUD_5224 := [[469.55, -29.1, 183.58], [0.102606, 0.699623, 0.706321, -0.033337], [0,0,0,0], [9E9, 9E9, 9E9, 9E9, 9E9, 9E9]];
	VAR robtarget OpenholeUD_5225 := [[465.57, -29.1, 183.19], [0.089791, 0.701383, 0.706823, -0.020014], [0,0,0,0], [9E9, 9E9, 9E9, 9E9, 9E9, 9E9]];
	VAR robtarget OpenholeUD_5226 := [[461.59, -29.1, 182.81], [0.076741, 0.70293, 0.707076, -0.006579], [0,0,0,0], [9E9, 9E9, 9E9, 9E9, 9E9, 9E9]];
	VAR robtarget OpenholeUD_5227 := [[457.61, -29.1, 182.42], [0.063492, 0.704251, 0.707073, 0.006925], [0,0,0,0], [9E9, 9E9, 9E9, 9E9, 9E9, 9E9]];
	VAR robtarget OpenholeUD_5228 := [[453.63, -29.1, 182.04], [0.050085, 0.705331, 0.706811, 0.020454], [0,0,0,0], [9E9, 9E9, 9E9, 9E9, 9E9, 9E9]];
	VAR robtarget OpenholeUD_5229 := [[449.65, -29.1, 181.65], [0.036561, 0.706161, 0.706291, 0.033965], [0,0,0,0], [9E9, 9E9, 9E9, 9E9, 9E9, 9E9]];
	VAR robtarget OpenholeUD_5230 := [[445.66, -29.1, 181.26], [0.022965, 0.706734, 0.705515, 0.047413], [0,0,0,0], [9E9, 9E9, 9E9, 9E9, 9E9, 9E9]];
	VAR robtarget OpenholeUD_5231 := [[441.68, -29.1, 180.88], [0.009342, 0.707045, 0.704492, 0.060755], [0,0,0,0], [9E9, 9E9, 9E9, 9E9, 9E9, 9E9]];
	VAR robtarget OpenholeUD_5232 := [[437.7, -29.1, 180.49], [-0.004263, 0.707094, 0.703229, 0.07395], [0,0,0,0], [9E9, 9E9, 9E9, 9E9, 9E9, 9E9]];
	VAR robtarget OpenholeUD_5233 := [[433.72, -29.1, 180.11], [-0.017803, 0.706883, 0.70174, 0.086957], [0,0,0,0], [9E9, 9E9, 9E9, 9E9, 9E9, 9E9]];
	VAR robtarget OpenholeUD_5234 := [[429.74, -29.1, 179.72], [-0.031236, 0.706417, 0.700037, 0.099743], [0,0,0,0], [9E9, 9E9, 9E9, 9E9, 9E9, 9E9]];
	VAR robtarget OpenholeUD_5235 := [[425.76, -29.1, 179.33], [-0.04452, 0.705704, 0.698137, 0.112273], [0,0,0,0], [9E9, 9E9, 9E9, 9E9, 9E9, 9E9]];
	VAR robtarget OpenholeUD_5236 := [[421.78, -29.1, 178.95], [-0.057617, 0.704755, 0.696057, 0.124519], [0,0,0,0], [9E9, 9E9, 9E9, 9E9, 9E9, 9E9]];
	VAR robtarget OpenholeUD_5237 := [[417.79, -29.1, 178.56], [-0.070492, 0.703584, 0.693815, 0.136457], [0,0,0,0], [9E9, 9E9, 9E9, 9E9, 9E9, 9E9]];
	VAR robtarget OpenholeUD_5238 := [[413.81, -29.1, 178.18], [-0.083114, 0.702205, 0.691431, 0.148066], [0,0,0,0], [9E9, 9E9, 9E9, 9E9, 9E9, 9E9]];
	VAR robtarget OpenholeUD_5239 := [[409.83, -29.1, 177.79], [-0.095455, 0.700634, 0.688922, 0.159331], [0,0,0,0], [9E9, 9E9, 9E9, 9E9, 9E9, 9E9]];
	VAR robtarget OpenholeUD_5240 := [[405.85, -29.1, 177.41], [-0.107492, 0.698889, 0.686308, 0.170239], [0,0,0,0], [9E9, 9E9, 9E9, 9E9, 9E9, 9E9]];
	VAR robtarget OpenholeUD_5241 := [[401.87, -29.1, 177.02], [-0.119208, 0.696986, 0.683607, 0.180782], [0,0,0,0], [9E9, 9E9, 9E9, 9E9, 9E9, 9E9]];
	VAR robtarget OpenholeUD_5242 := [[397.89, -29.1, 176.63], [-0.130586, 0.694944, 0.680835, 0.190955], [0,0,0,0], [9E9, 9E9, 9E9, 9E9, 9E9, 9E9]];
	VAR robtarget OpenholeUD_5243 := [[393.91, -29.1, 176.25], [-0.141617, 0.69278, 0.678009, 0.200757], [0,0,0,0], [9E9, 9E9, 9E9, 9E9, 9E9, 9E9]];
	VAR robtarget OpenholeUD_5244 := [[389.33, -29.1, 175.8], [-0.153863, 0.690164, 0.674713, 0.211571], [0,0,0,0], [9E9, 9E9, 9E9, 9E9, 9E9, 9E9]];
	VAR robtarget OpenholeUD_5245 := [[385.33, -29.1, 175.82], [-0.183051, 0.683002, 0.683002, 0.183051], [0,0,0,0], [9E9, 9E9, 9E9, 9E9, 9E9, 9E9]];
	VAR robtarget OpenholeUD_5246 := [[381.33, -29.1, 175.83], [-0.183051, 0.683002, 0.683002, 0.183051], [0,0,0,0], [9E9, 9E9, 9E9, 9E9, 9E9, 9E9]];
	VAR robtarget OpenholeUD_5247 := [[377.33, -29.1, 175.84], [-0.183051, 0.683002, 0.683002, 0.183051], [0,0,0,0], [9E9, 9E9, 9E9, 9E9, 9E9, 9E9]];
	VAR robtarget OpenholeUD_5248 := [[373.33, -29.1, 175.85], [-0.183051, 0.683002, 0.683002, 0.183051], [0,0,0,0], [9E9, 9E9, 9E9, 9E9, 9E9, 9E9]];
	VAR robtarget OpenholeUD_5249 := [[369.33, -29.1, 175.87], [-0.183051, 0.683002, 0.683002, 0.183051], [0,0,0,0], [9E9, 9E9, 9E9, 9E9, 9E9, 9E9]];
	VAR robtarget OpenholeUD_5250 := [[369.33, -29.1, 175.87], [-0.183051, 0.683002, 0.683002, 0.183051], [0,0,0,0], [9E9, 9E9, 9E9, 9E9, 9E9, 9E9]];
	VAR robtarget OpenholeUD_5251 := [[369.33, -30.3, 175.17], [-0.183051, 0.683002, 0.683002, 0.183051], [0,0,0,0], [9E9, 9E9, 9E9, 9E9, 9E9, 9E9]];
	VAR robtarget OpenholeUD_5252 := [[373.33, -30.3, 175.16], [-0.183051, 0.683002, 0.683002, 0.183051], [0,0,0,0], [9E9, 9E9, 9E9, 9E9, 9E9, 9E9]];
	VAR robtarget OpenholeUD_5253 := [[377.33, -30.3, 175.15], [-0.183051, 0.683002, 0.683002, 0.183051], [0,0,0,0], [9E9, 9E9, 9E9, 9E9, 9E9, 9E9]];
	VAR robtarget OpenholeUD_5254 := [[381.33, -30.3, 175.14], [-0.183051, 0.683002, 0.683002, 0.183051], [0,0,0,0], [9E9, 9E9, 9E9, 9E9, 9E9, 9E9]];
	VAR robtarget OpenholeUD_5255 := [[385.33, -30.3, 175.12], [-0.183051, 0.683002, 0.683002, 0.183051], [0,0,0,0], [9E9, 9E9, 9E9, 9E9, 9E9, 9E9]];
	VAR robtarget OpenholeUD_5256 := [[389.33, -30.3, 175.11], [-0.150428, 0.690921, 0.673656, 0.214912], [0,0,0,0], [9E9, 9E9, 9E9, 9E9, 9E9, 9E9]];
	VAR robtarget OpenholeUD_5257 := [[393.3, -30.3, 175.54], [-0.139752, 0.693159, 0.676552, 0.205615], [0,0,0,0], [9E9, 9E9, 9E9, 9E9, 9E9, 9E9]];
	VAR robtarget OpenholeUD_5258 := [[397.28, -30.3, 175.97], [-0.128722, 0.695292, 0.679415, 0.195948], [0,0,0,0], [9E9, 9E9, 9E9, 9E9, 9E9, 9E9]];
	VAR robtarget OpenholeUD_5259 := [[401.26, -30.3, 176.41], [-0.117345, 0.697302, 0.68223, 0.185909], [0,0,0,0], [9E9, 9E9, 9E9, 9E9, 9E9, 9E9]];
	VAR robtarget OpenholeUD_5260 := [[405.23, -30.3, 176.84], [-0.105634, 0.699172, 0.684982, 0.175499], [0,0,0,0], [9E9, 9E9, 9E9, 9E9, 9E9, 9E9]];
	VAR robtarget OpenholeUD_5261 := [[409.21, -30.3, 177.27], [-0.093601, 0.700884, 0.687653, 0.164721], [0,0,0,0], [9E9, 9E9, 9E9, 9E9, 9E9, 9E9]];
	VAR robtarget OpenholeUD_5262 := [[413.19, -30.3, 177.7], [-0.081267, 0.702421, 0.690226, 0.153583], [0,0,0,0], [9E9, 9E9, 9E9, 9E9, 9E9, 9E9]];
	VAR robtarget OpenholeUD_5263 := [[417.16, -30.3, 178.13], [-0.068652, 0.703766, 0.692683, 0.142095], [0,0,0,0], [9E9, 9E9, 9E9, 9E9, 9E9, 9E9]];
	VAR robtarget OpenholeUD_5264 := [[421.14, -30.3, 178.56], [-0.055786, 0.704903, 0.695003, 0.130272], [0,0,0,0], [9E9, 9E9, 9E9, 9E9, 9E9, 9E9]];
	VAR robtarget OpenholeUD_5265 := [[425.12, -30.3, 178.99], [-0.042698, 0.705816, 0.697169, 0.118134], [0,0,0,0], [9E9, 9E9, 9E9, 9E9, 9E9, 9E9]];
	VAR robtarget OpenholeUD_5266 := [[429.09, -30.3, 179.42], [-0.029423, 0.706494, 0.699162, 0.105703], [0,0,0,0], [9E9, 9E9, 9E9, 9E9, 9E9, 9E9]];
	VAR robtarget OpenholeUD_5267 := [[433.07, -30.3, 179.86], [-0.016, 0.706926, 0.700963, 0.093007], [0,0,0,0], [9E9, 9E9, 9E9, 9E9, 9E9, 9E9]];
	VAR robtarget OpenholeUD_5268 := [[437.05, -30.3, 180.29], [-0.002469, 0.707102, 0.702558, 0.080077], [0,0,0,0], [9E9, 9E9, 9E9, 9E9, 9E9, 9E9]];
	VAR robtarget OpenholeUD_5269 := [[441.02, -30.3, 180.72], [0.011126, 0.707019, 0.70393, 0.066948], [0,0,0,0], [9E9, 9E9, 9E9, 9E9, 9E9, 9E9]];
	VAR robtarget OpenholeUD_5270 := [[445, -30.3, 181.15], [0.024739, 0.706674, 0.705068, 0.053658], [0,0,0,0], [9E9, 9E9, 9E9, 9E9, 9E9, 9E9]];
	VAR robtarget OpenholeUD_5271 := [[448.98, -30.3, 181.58], [0.038326, 0.706067, 0.70596, 0.040249], [0,0,0,0], [9E9, 9E9, 9E9, 9E9, 9E9, 9E9]];
	VAR robtarget OpenholeUD_5272 := [[452.95, -30.3, 182.01], [0.051842, 0.705204, 0.7066, 0.026763], [0,0,0,0], [9E9, 9E9, 9E9, 9E9, 9E9, 9E9]];
	VAR robtarget OpenholeUD_5273 := [[456.93, -30.3, 182.44], [0.065241, 0.704091, 0.706983, 0.013243], [0,0,0,0], [9E9, 9E9, 9E9, 9E9, 9E9, 9E9]];
	VAR robtarget OpenholeUD_5274 := [[460.91, -30.3, 182.88], [0.078482, 0.702738, 0.707107, -0.000265], [0,0,0,0], [9E9, 9E9, 9E9, 9E9, 9E9, 9E9]];
	VAR robtarget OpenholeUD_5275 := [[464.88, -30.3, 183.31], [0.091524, 0.701159, 0.706974, -0.013719], [0,0,0,0], [9E9, 9E9, 9E9, 9E9, 9E9, 9E9]];
	VAR robtarget OpenholeUD_5276 := [[468.86, -30.3, 183.74], [0.104333, 0.699367, 0.706588, -0.027075], [0,0,0,0], [9E9, 9E9, 9E9, 9E9, 9E9, 9E9]];
	VAR robtarget OpenholeUD_5277 := [[472.84, -30.3, 184.17], [0.116874, 0.697381, 0.705958, -0.040293], [0,0,0,0], [9E9, 9E9, 9E9, 9E9, 9E9, 9E9]];
	VAR robtarget OpenholeUD_5278 := [[476.81, -30.3, 184.6], [0.12912, 0.695218, 0.705092, -0.053336], [0,0,0,0], [9E9, 9E9, 9E9, 9E9, 9E9, 9E9]];
	VAR robtarget OpenholeUD_5279 := [[480.79, -30.3, 185.03], [0.141046, 0.692897, 0.704004, -0.066168], [0,0,0,0], [9E9, 9E9, 9E9, 9E9, 9E9, 9E9]];
	VAR robtarget OpenholeUD_5280 := [[484.77, -30.3, 185.46], [0.152633, 0.690437, 0.702707, -0.078758], [0,0,0,0], [9E9, 9E9, 9E9, 9E9, 9E9, 9E9]];
	VAR robtarget OpenholeUD_5281 := [[488.74, -30.3, 185.89], [0.163865, 0.687858, 0.701216, -0.09108], [0,0,0,0], [9E9, 9E9, 9E9, 9E9, 9E9, 9E9]];
	VAR robtarget OpenholeUD_5282 := [[492.72, -30.3, 186.33], [0.17473, 0.685178, 0.699549, -0.103109], [0,0,0,0], [9E9, 9E9, 9E9, 9E9, 9E9, 9E9]];
	VAR robtarget OpenholeUD_5283 := [[496.7, -30.3, 186.76], [0.185223, 0.682417, 0.697721, -0.114828], [0,0,0,0], [9E9, 9E9, 9E9, 9E9, 9E9, 9E9]];
	VAR robtarget OpenholeUD_5284 := [[500.67, -30.3, 187.19], [0.195338, 0.67959, 0.69575, -0.12622], [0,0,0,0], [9E9, 9E9, 9E9, 9E9, 9E9, 9E9]];
	VAR robtarget OpenholeUD_5285 := [[504.65, -30.3, 187.62], [0.205075, 0.676716, 0.693654, -0.137273], [0,0,0,0], [9E9, 9E9, 9E9, 9E9, 9E9, 9E9]];
	VAR robtarget OpenholeUD_5286 := [[509.37, -30.3, 188.13], [0.183051, 0.683002, 0.683002, -0.183051], [0,0,0,0], [9E9, 9E9, 9E9, 9E9, 9E9, 9E9]];
	VAR robtarget OpenholeUD_5287 := [[513.37, -30.3, 188.12], [0.183051, 0.683002, 0.683002, -0.183051], [0,0,0,0], [9E9, 9E9, 9E9, 9E9, 9E9, 9E9]];
	VAR robtarget OpenholeUD_5288 := [[517.37, -30.3, 188.11], [0.183051, 0.683002, 0.683002, -0.183051], [0,0,0,0], [9E9, 9E9, 9E9, 9E9, 9E9, 9E9]];
	VAR robtarget OpenholeUD_5289 := [[521.37, -30.3, 188.09], [0.183051, 0.683002, 0.683002, -0.183051], [0,0,0,0], [9E9, 9E9, 9E9, 9E9, 9E9, 9E9]];
	VAR robtarget OpenholeUD_5290 := [[525.37, -30.3, 188.08], [0.183051, 0.683002, 0.683002, -0.183051], [0,0,0,0], [9E9, 9E9, 9E9, 9E9, 9E9, 9E9]];
	VAR robtarget OpenholeUD_5291 := [[529.37, -30.3, 188.07], [0.183051, 0.683002, 0.683002, -0.183051], [0,0,0,0], [9E9, 9E9, 9E9, 9E9, 9E9, 9E9]];
	VAR robtarget OpenholeUD_5292 := [[529.37, -30.3, 188.07], [0.183051, 0.683002, 0.683002, -0.183051], [0,0,0,0], [9E9, 9E9, 9E9, 9E9, 9E9, 9E9]];
	VAR robtarget OpenholeUD_5293 := [[529.37, -31.5, 188.76], [0.183051, 0.683002, 0.683002, -0.183051], [0,0,0,0], [9E9, 9E9, 9E9, 9E9, 9E9, 9E9]];
	VAR robtarget OpenholeUD_5294 := [[525.37, -31.5, 188.77], [0.183051, 0.683002, 0.683002, -0.183051], [0,0,0,0], [9E9, 9E9, 9E9, 9E9, 9E9, 9E9]];
	VAR robtarget OpenholeUD_5295 := [[521.37, -31.5, 188.79], [0.183051, 0.683002, 0.683002, -0.183051], [0,0,0,0], [9E9, 9E9, 9E9, 9E9, 9E9, 9E9]];
	VAR robtarget OpenholeUD_5296 := [[517.37, -31.5, 188.8], [0.183051, 0.683002, 0.683002, -0.183051], [0,0,0,0], [9E9, 9E9, 9E9, 9E9, 9E9, 9E9]];
	VAR robtarget OpenholeUD_5297 := [[513.37, -31.5, 188.81], [0.183051, 0.683002, 0.683002, -0.183051], [0,0,0,0], [9E9, 9E9, 9E9, 9E9, 9E9, 9E9]];
	VAR robtarget OpenholeUD_5298 := [[509.37, -31.5, 188.82], [0.183051, 0.683002, 0.683002, -0.183051], [0,0,0,0], [9E9, 9E9, 9E9, 9E9, 9E9, 9E9]];
	VAR robtarget OpenholeUD_5299 := [[505.4, -31.5, 188.35], [0.210264, 0.675121, 0.693937, -0.135835], [0,0,0,0], [9E9, 9E9, 9E9, 9E9, 9E9, 9E9]];
	VAR robtarget OpenholeUD_5300 := [[501.43, -31.5, 187.87], [0.200679, 0.678033, 0.696007, -0.124796], [0,0,0,0], [9E9, 9E9, 9E9, 9E9, 9E9, 9E9]];
	VAR robtarget OpenholeUD_5301 := [[497.46, -31.5, 187.4], [0.190715, 0.680902, 0.697951, -0.113421], [0,0,0,0], [9E9, 9E9, 9E9, 9E9, 9E9, 9E9]];
	VAR robtarget OpenholeUD_5302 := [[493.48, -31.5, 186.92], [0.180373, 0.683715, 0.699752, -0.10172], [0,0,0,0], [9E9, 9E9, 9E9, 9E9, 9E9, 9E9]];
	VAR robtarget OpenholeUD_5303 := [[489.51, -31.5, 186.44], [0.169655, 0.686453, 0.701393, -0.089708], [0,0,0,0], [9E9, 9E9, 9E9, 9E9, 9E9, 9E9]];
	VAR robtarget OpenholeUD_5304 := [[485.54, -31.5, 185.97], [0.158567, 0.689098, 0.702857, -0.077405], [0,0,0,0], [9E9, 9E9, 9E9, 9E9, 9E9, 9E9]];
	VAR robtarget OpenholeUD_5305 := [[481.57, -31.5, 185.49], [0.14712, 0.691633, 0.704128, -0.064832], [0,0,0,0], [9E9, 9E9, 9E9, 9E9, 9E9, 9E9]];
	VAR robtarget OpenholeUD_5306 := [[477.6, -31.5, 185.01], [0.135326, 0.694037, 0.705191, -0.052018], [0,0,0,0], [9E9, 9E9, 9E9, 9E9, 9E9, 9E9]];
	VAR robtarget OpenholeUD_5307 := [[473.63, -31.5, 184.54], [0.123205, 0.696291, 0.706031, -0.038993], [0,0,0,0], [9E9, 9E9, 9E9, 9E9, 9E9, 9E9]];
	VAR robtarget OpenholeUD_5308 := [[469.66, -31.5, 184.06], [0.110779, 0.698375, 0.706636, -0.025791], [0,0,0,0], [9E9, 9E9, 9E9, 9E9, 9E9, 9E9]];
	VAR robtarget OpenholeUD_5309 := [[465.68, -31.5, 183.58], [0.098075, 0.700272, 0.706997, -0.012449], [0,0,0,0], [9E9, 9E9, 9E9, 9E9, 9E9, 9E9]];
	VAR robtarget OpenholeUD_5310 := [[461.71, -31.5, 183.11], [0.085124, 0.701964, 0.707106, 0.000991], [0,0,0,0], [9E9, 9E9, 9E9, 9E9, 9E9, 9E9]];
	VAR robtarget OpenholeUD_5311 := [[457.74, -31.5, 182.63], [0.071961, 0.703436, 0.706958, 0.014488], [0,0,0,0], [9E9, 9E9, 9E9, 9E9, 9E9, 9E9]];
	VAR robtarget OpenholeUD_5312 := [[453.77, -31.5, 182.15], [0.058625, 0.704672, 0.706552, 0.027998], [0,0,0,0], [9E9, 9E9, 9E9, 9E9, 9E9, 9E9]];
	VAR robtarget OpenholeUD_5313 := [[449.8, -31.5, 181.68], [0.045158, 0.705663, 0.705889, 0.041478], [0,0,0,0], [9E9, 9E9, 9E9, 9E9, 9E9, 9E9]];
	VAR robtarget OpenholeUD_5314 := [[445.83, -31.5, 181.2], [0.031602, 0.7064, 0.704974, 0.054882], [0,0,0,0], [9E9, 9E9, 9E9, 9E9, 9E9, 9E9]];
	VAR robtarget OpenholeUD_5315 := [[441.85, -31.5, 180.72], [0.018004, 0.706878, 0.703813, 0.068168], [0,0,0,0], [9E9, 9E9, 9E9, 9E9, 9E9, 9E9]];
	VAR robtarget OpenholeUD_5316 := [[437.88, -31.5, 180.25], [0.004408, 0.707093, 0.702418, 0.081296], [0,0,0,0], [9E9, 9E9, 9E9, 9E9, 9E9, 9E9]];
	VAR robtarget OpenholeUD_5317 := [[433.91, -31.5, 179.77], [-0.009141, 0.707048, 0.7008, 0.094227], [0,0,0,0], [9E9, 9E9, 9E9, 9E9, 9E9, 9E9]];
	VAR robtarget OpenholeUD_5318 := [[429.94, -31.5, 179.29], [-0.022599, 0.706746, 0.698976, 0.106925], [0,0,0,0], [9E9, 9E9, 9E9, 9E9, 9E9, 9E9]];
	VAR robtarget OpenholeUD_5319 := [[425.97, -31.5, 178.82], [-0.035923, 0.706194, 0.69696, 0.11936], [0,0,0,0], [9E9, 9E9, 9E9, 9E9, 9E9, 9E9]];
	VAR robtarget OpenholeUD_5320 := [[422, -31.5, 178.34], [-0.049075, 0.705402, 0.694771, 0.131503], [0,0,0,0], [9E9, 9E9, 9E9, 9E9, 9E9, 9E9]];
	VAR robtarget OpenholeUD_5321 := [[418.03, -31.5, 177.86], [-0.062019, 0.704382, 0.692428, 0.143331], [0,0,0,0], [9E9, 9E9, 9E9, 9E9, 9E9, 9E9]];
	VAR robtarget OpenholeUD_5322 := [[414.05, -31.5, 177.39], [-0.074722, 0.703148, 0.689949, 0.154824], [0,0,0,0], [9E9, 9E9, 9E9, 9E9, 9E9, 9E9]];
	VAR robtarget OpenholeUD_5323 := [[410.08, -31.5, 176.91], [-0.087157, 0.701715, 0.687353, 0.165968], [0,0,0,0], [9E9, 9E9, 9E9, 9E9, 9E9, 9E9]];
	VAR robtarget OpenholeUD_5324 := [[406.11, -31.5, 176.43], [-0.099298, 0.7001, 0.68466, 0.176752], [0,0,0,0], [9E9, 9E9, 9E9, 9E9, 9E9, 9E9]];
	VAR robtarget OpenholeUD_5325 := [[402.14, -31.5, 175.96], [-0.111127, 0.69832, 0.681886, 0.187168], [0,0,0,0], [9E9, 9E9, 9E9, 9E9, 9E9, 9E9]];
	VAR robtarget OpenholeUD_5326 := [[398.17, -31.5, 175.48], [-0.122626, 0.696393, 0.679049, 0.197212], [0,0,0,0], [9E9, 9E9, 9E9, 9E9, 9E9, 9E9]];
	VAR robtarget OpenholeUD_5327 := [[394.2, -31.5, 175], [-0.133785, 0.694335, 0.676165, 0.206883], [0,0,0,0], [9E9, 9E9, 9E9, 9E9, 9E9, 9E9]];
	VAR robtarget OpenholeUD_5328 := [[389.32, -31.5, 174.42], [-0.146996, 0.691659, 0.672585, 0.218242], [0,0,0,0], [9E9, 9E9, 9E9, 9E9, 9E9, 9E9]];
	VAR robtarget OpenholeUD_5329 := [[385.32, -31.5, 174.43], [-0.183051, 0.683002, 0.683002, 0.183051], [0,0,0,0], [9E9, 9E9, 9E9, 9E9, 9E9, 9E9]];
	VAR robtarget OpenholeUD_5330 := [[381.32, -31.5, 174.44], [-0.183051, 0.683002, 0.683002, 0.183051], [0,0,0,0], [9E9, 9E9, 9E9, 9E9, 9E9, 9E9]];
	VAR robtarget OpenholeUD_5331 := [[377.32, -31.5, 174.46], [-0.183051, 0.683002, 0.683002, 0.183051], [0,0,0,0], [9E9, 9E9, 9E9, 9E9, 9E9, 9E9]];
	VAR robtarget OpenholeUD_5332 := [[373.32, -31.5, 174.47], [-0.183051, 0.683002, 0.683002, 0.183051], [0,0,0,0], [9E9, 9E9, 9E9, 9E9, 9E9, 9E9]];
	VAR robtarget OpenholeUD_5333 := [[369.32, -31.5, 174.48], [-0.183051, 0.683002, 0.683002, 0.183051], [0,0,0,0], [9E9, 9E9, 9E9, 9E9, 9E9, 9E9]];
	VAR robtarget OpenholeUD_5334 := [[369.32, -31.5, 174.48], [-0.183051, 0.683002, 0.683002, 0.183051], [0,0,0,0], [9E9, 9E9, 9E9, 9E9, 9E9, 9E9]];
	VAR robtarget OpenholeUD_5335 := [[369.32, -32.7, 173.79], [-0.183051, 0.683002, 0.683002, 0.183051], [0,0,0,0], [9E9, 9E9, 9E9, 9E9, 9E9, 9E9]];
	VAR robtarget OpenholeUD_5336 := [[373.32, -32.7, 173.78], [-0.183051, 0.683002, 0.683002, 0.183051], [0,0,0,0], [9E9, 9E9, 9E9, 9E9, 9E9, 9E9]];
	VAR robtarget OpenholeUD_5337 := [[377.32, -32.7, 173.76], [-0.183051, 0.683002, 0.683002, 0.183051], [0,0,0,0], [9E9, 9E9, 9E9, 9E9, 9E9, 9E9]];
	VAR robtarget OpenholeUD_5338 := [[381.32, -32.7, 173.75], [-0.183051, 0.683002, 0.683002, 0.183051], [0,0,0,0], [9E9, 9E9, 9E9, 9E9, 9E9, 9E9]];
	VAR robtarget OpenholeUD_5339 := [[385.32, -32.7, 173.74], [-0.183051, 0.683002, 0.683002, 0.183051], [0,0,0,0], [9E9, 9E9, 9E9, 9E9, 9E9, 9E9]];
	VAR robtarget OpenholeUD_5340 := [[389.32, -32.7, 173.72], [-0.143568, 0.692379, 0.671499, 0.22156], [0,0,0,0], [9E9, 9E9, 9E9, 9E9, 9E9, 9E9]];
	VAR robtarget OpenholeUD_5341 := [[393.29, -32.7, 174.25], [-0.132788, 0.694527, 0.674445, 0.212423], [0,0,0,0], [9E9, 9E9, 9E9, 9E9, 9E9, 9E9]];
	VAR robtarget OpenholeUD_5342 := [[397.25, -32.7, 174.77], [-0.121661, 0.696562, 0.677366, 0.202917], [0,0,0,0], [9E9, 9E9, 9E9, 9E9, 9E9, 9E9]];
	VAR robtarget OpenholeUD_5343 := [[401.22, -32.7, 175.29], [-0.110193, 0.698468, 0.680247, 0.193039], [0,0,0,0], [9E9, 9E9, 9E9, 9E9, 9E9, 9E9]];
	VAR robtarget OpenholeUD_5344 := [[405.19, -32.7, 175.81], [-0.098397, 0.700227, 0.683073, 0.182787], [0,0,0,0], [9E9, 9E9, 9E9, 9E9, 9E9, 9E9]];
	VAR robtarget OpenholeUD_5345 := [[409.15, -32.7, 176.33], [-0.086288, 0.701822, 0.685828, 0.172164], [0,0,0,0], [9E9, 9E9, 9E9, 9E9, 9E9, 9E9]];
	VAR robtarget OpenholeUD_5346 := [[413.12, -32.7, 176.86], [-0.073885, 0.703236, 0.688492, 0.161178], [0,0,0,0], [9E9, 9E9, 9E9, 9E9, 9E9, 9E9]];
	VAR robtarget OpenholeUD_5347 := [[417.08, -32.7, 177.38], [-0.061212, 0.704452, 0.691049, 0.149836], [0,0,0,0], [9E9, 9E9, 9E9, 9E9, 9E9, 9E9]];
	VAR robtarget OpenholeUD_5348 := [[421.05, -32.7, 177.9], [-0.048298, 0.705455, 0.693479, 0.138153], [0,0,0,0], [9E9, 9E9, 9E9, 9E9, 9E9, 9E9]];
	VAR robtarget OpenholeUD_5349 := [[425.01, -32.7, 178.42], [-0.035173, 0.706231, 0.695764, 0.126146], [0,0,0,0], [9E9, 9E9, 9E9, 9E9, 9E9, 9E9]];
	VAR robtarget OpenholeUD_5350 := [[428.98, -32.7, 178.94], [-0.021873, 0.706768, 0.697883, 0.113838], [0,0,0,0], [9E9, 9E9, 9E9, 9E9, 9E9, 9E9]];
	VAR robtarget OpenholeUD_5351 := [[432.95, -32.7, 179.46], [-0.008437, 0.707056, 0.69982, 0.101254], [0,0,0,0], [9E9, 9E9, 9E9, 9E9, 9E9, 9E9]];
	VAR robtarget OpenholeUD_5352 := [[436.91, -32.7, 179.99], [0.005094, 0.707088, 0.701556, 0.088424], [0,0,0,0], [9E9, 9E9, 9E9, 9E9, 9E9, 9E9]];
	VAR robtarget OpenholeUD_5353 := [[440.88, -32.7, 180.51], [0.018676, 0.70686, 0.703077, 0.075382], [0,0,0,0], [9E9, 9E9, 9E9, 9E9, 9E9, 9E9]];
	VAR robtarget OpenholeUD_5354 := [[444.84, -32.7, 181.03], [0.032265, 0.70637, 0.704369, 0.062166], [0,0,0,0], [9E9, 9E9, 9E9, 9E9, 9E9, 9E9]];
	VAR robtarget OpenholeUD_5355 := [[448.81, -32.7, 181.55], [0.045815, 0.705621, 0.70542, 0.048816], [0,0,0,0], [9E9, 9E9, 9E9, 9E9, 9E9, 9E9]];
	VAR robtarget OpenholeUD_5356 := [[452.78, -32.7, 182.07], [0.05928, 0.704618, 0.706221, 0.035372], [0,0,0,0], [9E9, 9E9, 9E9, 9E9, 9E9, 9E9]];
	VAR robtarget OpenholeUD_5357 := [[456.74, -32.7, 182.59], [0.072618, 0.703368, 0.706768, 0.02188], [0,0,0,0], [9E9, 9E9, 9E9, 9E9, 9E9, 9E9]];
	VAR robtarget OpenholeUD_5358 := [[460.71, -32.7, 183.12], [0.085787, 0.701884, 0.707057, 0.008383], [0,0,0,0], [9E9, 9E9, 9E9, 9E9, 9E9, 9E9]];
	VAR robtarget OpenholeUD_5359 := [[464.67, -32.7, 183.64], [0.098748, 0.700178, 0.707089, -0.005075], [0,0,0,0], [9E9, 9E9, 9E9, 9E9, 9E9, 9E9]];
	VAR robtarget OpenholeUD_5360 := [[468.64, -32.7, 184.16], [0.111465, 0.698266, 0.706866, -0.018451], [0,0,0,0], [9E9, 9E9, 9E9, 9E9, 9E9, 9E9]];
	VAR robtarget OpenholeUD_5361 := [[472.6, -32.7, 184.68], [0.123906, 0.696166, 0.706396, -0.031704], [0,0,0,0], [9E9, 9E9, 9E9, 9E9, 9E9, 9E9]];
	VAR robtarget OpenholeUD_5362 := [[476.57, -32.7, 185.2], [0.136045, 0.693896, 0.705686, -0.044797], [0,0,0,0], [9E9, 9E9, 9E9, 9E9, 9E9, 9E9]];
	VAR robtarget OpenholeUD_5363 := [[480.54, -32.7, 185.72], [0.147858, 0.691475, 0.704749, -0.057693], [0,0,0,0], [9E9, 9E9, 9E9, 9E9, 9E9, 9E9]];
	VAR robtarget OpenholeUD_5364 := [[484.5, -32.7, 186.25], [0.159326, 0.688923, 0.703598, -0.070359], [0,0,0,0], [9E9, 9E9, 9E9, 9E9, 9E9, 9E9]];
	VAR robtarget OpenholeUD_5365 := [[488.47, -32.7, 186.77], [0.170435, 0.686259, 0.702246, -0.082769], [0,0,0,0], [9E9, 9E9, 9E9, 9E9, 9E9, 9E9]];
	VAR robtarget OpenholeUD_5366 := [[492.43, -32.7, 187.29], [0.181174, 0.683503, 0.70071, -0.094897], [0,0,0,0], [9E9, 9E9, 9E9, 9E9, 9E9, 9E9]];
	VAR robtarget OpenholeUD_5367 := [[496.4, -32.7, 187.81], [0.191538, 0.680671, 0.699006, -0.106724], [0,0,0,0], [9E9, 9E9, 9E9, 9E9, 9E9, 9E9]];
	VAR robtarget OpenholeUD_5368 := [[500.37, -32.7, 188.33], [0.201523, 0.677782, 0.697152, -0.118231], [0,0,0,0], [9E9, 9E9, 9E9, 9E9, 9E9, 9E9]];
	VAR robtarget OpenholeUD_5369 := [[504.33, -32.7, 188.85], [0.211129, 0.674852, 0.695164, -0.129408], [0,0,0,0], [9E9, 9E9, 9E9, 9E9, 9E9, 9E9]];
	VAR robtarget OpenholeUD_5370 := [[509.37, -32.7, 189.52], [0.183051, 0.683002, 0.683002, -0.183051], [0,0,0,0], [9E9, 9E9, 9E9, 9E9, 9E9, 9E9]];
	VAR robtarget OpenholeUD_5371 := [[513.37, -32.7, 189.51], [0.183051, 0.683002, 0.683002, -0.183051], [0,0,0,0], [9E9, 9E9, 9E9, 9E9, 9E9, 9E9]];
	VAR robtarget OpenholeUD_5372 := [[517.37, -32.7, 189.49], [0.183051, 0.683002, 0.683002, -0.183051], [0,0,0,0], [9E9, 9E9, 9E9, 9E9, 9E9, 9E9]];
	VAR robtarget OpenholeUD_5373 := [[521.37, -32.7, 189.48], [0.183051, 0.683002, 0.683002, -0.183051], [0,0,0,0], [9E9, 9E9, 9E9, 9E9, 9E9, 9E9]];
	VAR robtarget OpenholeUD_5374 := [[525.37, -32.7, 189.47], [0.183051, 0.683002, 0.683002, -0.183051], [0,0,0,0], [9E9, 9E9, 9E9, 9E9, 9E9, 9E9]];
	VAR robtarget OpenholeUD_5375 := [[529.37, -32.7, 189.46], [0.183051, 0.683002, 0.683002, -0.183051], [0,0,0,0], [9E9, 9E9, 9E9, 9E9, 9E9, 9E9]];
	VAR robtarget OpenholeUD_5376 := [[529.37, -32.7, 189.46], [0.183051, 0.683002, 0.683002, -0.183051], [0,0,0,0], [9E9, 9E9, 9E9, 9E9, 9E9, 9E9]];
	VAR robtarget OpenholeUD_5377 := [[529.37, -33.9, 190.15], [0.183051, 0.683002, 0.683002, -0.183051], [0,0,0,0], [9E9, 9E9, 9E9, 9E9, 9E9, 9E9]];
	VAR robtarget OpenholeUD_5378 := [[525.37, -33.9, 190.16], [0.183051, 0.683002, 0.683002, -0.183051], [0,0,0,0], [9E9, 9E9, 9E9, 9E9, 9E9, 9E9]];
	VAR robtarget OpenholeUD_5379 := [[521.37, -33.9, 190.17], [0.183051, 0.683002, 0.683002, -0.183051], [0,0,0,0], [9E9, 9E9, 9E9, 9E9, 9E9, 9E9]];
	VAR robtarget OpenholeUD_5380 := [[517.37, -33.9, 190.19], [0.183051, 0.683002, 0.683002, -0.183051], [0,0,0,0], [9E9, 9E9, 9E9, 9E9, 9E9, 9E9]];
	VAR robtarget OpenholeUD_5381 := [[513.37, -33.9, 190.2], [0.183051, 0.683002, 0.683002, -0.183051], [0,0,0,0], [9E9, 9E9, 9E9, 9E9, 9E9, 9E9]];
	VAR robtarget OpenholeUD_5382 := [[509.37, -33.9, 190.21], [0.183051, 0.683002, 0.683002, -0.183051], [0,0,0,0], [9E9, 9E9, 9E9, 9E9, 9E9, 9E9]];
	VAR robtarget OpenholeUD_5383 := [[505.41, -33.9, 189.64], [0.217059, 0.672968, 0.695253, -0.128932], [0,0,0,0], [9E9, 9E9, 9E9, 9E9, 9E9, 9E9]];
	VAR robtarget OpenholeUD_5384 := [[501.46, -33.9, 189.08], [0.207638, 0.675934, 0.697225, -0.117802], [0,0,0,0], [9E9, 9E9, 9E9, 9E9, 9E9, 9E9]];
	VAR robtarget OpenholeUD_5385 := [[497.5, -33.9, 188.51], [0.197839, 0.678866, 0.699065, -0.106342], [0,0,0,0], [9E9, 9E9, 9E9, 9E9, 9E9, 9E9]];
	VAR robtarget OpenholeUD_5386 := [[493.54, -33.9, 187.94], [0.18766, 0.68175, 0.700755, -0.094563], [0,0,0,0], [9E9, 9E9, 9E9, 9E9, 9E9, 9E9]];
	VAR robtarget OpenholeUD_5387 := [[489.58, -33.9, 187.38], [0.177103, 0.684569, 0.70228, -0.082481], [0,0,0,0], [9E9, 9E9, 9E9, 9E9, 9E9, 9E9]];
	VAR robtarget OpenholeUD_5388 := [[485.62, -33.9, 186.81], [0.166173, 0.687304, 0.703622, -0.070115], [0,0,0,0], [9E9, 9E9, 9E9, 9E9, 9E9, 9E9]];
	VAR robtarget OpenholeUD_5389 := [[481.66, -33.9, 186.24], [0.154878, 0.689937, 0.704766, -0.05749], [0,0,0,0], [9E9, 9E9, 9E9, 9E9, 9E9, 9E9]];
	VAR robtarget OpenholeUD_5390 := [[477.7, -33.9, 185.68], [0.143231, 0.692448, 0.705697, -0.044634], [0,0,0,0], [9E9, 9E9, 9E9, 9E9, 9E9, 9E9]];
	VAR robtarget OpenholeUD_5391 := [[473.74, -33.9, 185.11], [0.131249, 0.694819, 0.706401, -0.031577], [0,0,0,0], [9E9, 9E9, 9E9, 9E9, 9E9, 9E9]];
	VAR robtarget OpenholeUD_5392 := [[469.78, -33.9, 184.54], [0.118953, 0.69703, 0.706869, -0.018354], [0,0,0,0], [9E9, 9E9, 9E9, 9E9, 9E9, 9E9]];
	VAR robtarget OpenholeUD_5393 := [[465.82, -33.9, 183.98], [0.106369, 0.699061, 0.707089, -0.005004], [0,0,0,0], [9E9, 9E9, 9E9, 9E9, 9E9, 9E9]];
	VAR robtarget OpenholeUD_5394 := [[461.86, -33.9, 183.41], [0.093526, 0.700894, 0.707056, 0.008434], [0,0,0,0], [9E9, 9E9, 9E9, 9E9, 9E9, 9E9]];
	VAR robtarget OpenholeUD_5395 := [[457.9, -33.9, 182.85], [0.080459, 0.702514, 0.706767, 0.021916], [0,0,0,0], [9E9, 9E9, 9E9, 9E9, 9E9, 9E9]];
	VAR robtarget OpenholeUD_5396 := [[453.94, -33.9, 182.28], [0.067205, 0.703906, 0.70622, 0.035399], [0,0,0,0], [9E9, 9E9, 9E9, 9E9, 9E9, 9E9]];
	VAR robtarget OpenholeUD_5397 := [[449.98, -33.9, 181.71], [0.053804, 0.705057, 0.705418, 0.04884], [0,0,0,0], [9E9, 9E9, 9E9, 9E9, 9E9, 9E9]];
	VAR robtarget OpenholeUD_5398 := [[446.02, -33.9, 181.15], [0.0403, 0.705957, 0.704366, 0.062194], [0,0,0,0], [9E9, 9E9, 9E9, 9E9, 9E9, 9E9]];
	VAR robtarget OpenholeUD_5399 := [[442.06, -33.9, 180.58], [0.026736, 0.706601, 0.703073, 0.075419], [0,0,0,0], [9E9, 9E9, 9E9, 9E9, 9E9, 9E9]];
	VAR robtarget OpenholeUD_5400 := [[438.1, -33.9, 180.01], [0.013159, 0.706984, 0.70155, 0.088476], [0,0,0,0], [9E9, 9E9, 9E9, 9E9, 9E9, 9E9]];
	VAR robtarget OpenholeUD_5401 := [[434.14, -33.9, 179.45], [-0.000388, 0.707107, 0.699809, 0.101326], [0,0,0,0], [9E9, 9E9, 9E9, 9E9, 9E9, 9E9]];
	VAR robtarget OpenholeUD_5402 := [[430.18, -33.9, 178.88], [-0.01386, 0.706971, 0.697867, 0.113934], [0,0,0,0], [9E9, 9E9, 9E9, 9E9, 9E9, 9E9]];
	VAR robtarget OpenholeUD_5403 := [[426.22, -33.9, 178.31], [-0.027215, 0.706583, 0.695741, 0.126271], [0,0,0,0], [9E9, 9E9, 9E9, 9E9, 9E9, 9E9]];
	VAR robtarget OpenholeUD_5404 := [[422.26, -33.9, 177.75], [-0.040413, 0.705951, 0.693448, 0.13831], [0,0,0,0], [9E9, 9E9, 9E9, 9E9, 9E9, 9E9]];
	VAR robtarget OpenholeUD_5405 := [[418.3, -33.9, 177.18], [-0.053417, 0.705086, 0.691008, 0.150027], [0,0,0,0], [9E9, 9E9, 9E9, 9E9, 9E9, 9E9]];
	VAR robtarget OpenholeUD_5406 := [[414.34, -33.9, 176.61], [-0.066194, 0.704002, 0.688439, 0.161405], [0,0,0,0], [9E9, 9E9, 9E9, 9E9, 9E9, 9E9]];
	VAR robtarget OpenholeUD_5407 := [[410.38, -33.9, 176.05], [-0.078714, 0.702712, 0.685761, 0.17243], [0,0,0,0], [9E9, 9E9, 9E9, 9E9, 9E9, 9E9]];
	VAR robtarget OpenholeUD_5408 := [[406.42, -33.9, 175.48], [-0.090952, 0.701233, 0.682992, 0.18309], [0,0,0,0], [9E9, 9E9, 9E9, 9E9, 9E9, 9E9]];
	VAR robtarget OpenholeUD_5409 := [[402.46, -33.9, 174.91], [-0.102888, 0.699581, 0.68015, 0.19338], [0,0,0,0], [9E9, 9E9, 9E9, 9E9, 9E9, 9E9]];
	VAR robtarget OpenholeUD_5410 := [[398.5, -33.9, 174.35], [-0.114503, 0.697774, 0.677252, 0.203297], [0,0,0,0], [9E9, 9E9, 9E9, 9E9, 9E9, 9E9]];
	VAR robtarget OpenholeUD_5411 := [[394.54, -33.9, 173.78], [-0.125785, 0.695829, 0.674314, 0.21284], [0,0,0,0], [9E9, 9E9, 9E9, 9E9, 9E9, 9E9]];
	VAR robtarget OpenholeUD_5412 := [[389.32, -33.9, 173.03], [-0.140143, 0.69308, 0.6704, 0.224865], [0,0,0,0], [9E9, 9E9, 9E9, 9E9, 9E9, 9E9]];
	VAR robtarget OpenholeUD_5413 := [[385.32, -33.9, 173.04], [-0.183051, 0.683002, 0.683002, 0.183051], [0,0,0,0], [9E9, 9E9, 9E9, 9E9, 9E9, 9E9]];
	VAR robtarget OpenholeUD_5414 := [[381.32, -33.9, 173.06], [-0.183051, 0.683002, 0.683002, 0.183051], [0,0,0,0], [9E9, 9E9, 9E9, 9E9, 9E9, 9E9]];
	VAR robtarget OpenholeUD_5415 := [[377.32, -33.9, 173.07], [-0.183051, 0.683002, 0.683002, 0.183051], [0,0,0,0], [9E9, 9E9, 9E9, 9E9, 9E9, 9E9]];
	VAR robtarget OpenholeUD_5416 := [[373.32, -33.9, 173.08], [-0.183051, 0.683002, 0.683002, 0.183051], [0,0,0,0], [9E9, 9E9, 9E9, 9E9, 9E9, 9E9]];
	VAR robtarget OpenholeUD_5417 := [[369.32, -33.9, 173.09], [-0.183051, 0.683002, 0.683002, 0.183051], [0,0,0,0], [9E9, 9E9, 9E9, 9E9, 9E9, 9E9]];
	VAR robtarget OpenholeUD_5418 := [[369.32, -33.9, 173.09], [-0.183051, 0.683002, 0.683002, 0.183051], [0,0,0,0], [9E9, 9E9, 9E9, 9E9, 9E9, 9E9]];
	VAR robtarget OpenholeUD_5419 := [[369.32, -35.1, 172.4], [-0.183051, 0.683002, 0.683002, 0.183051], [0,0,0,0], [9E9, 9E9, 9E9, 9E9, 9E9, 9E9]];
	VAR robtarget OpenholeUD_5420 := [[373.32, -35.1, 172.39], [-0.183051, 0.683002, 0.683002, 0.183051], [0,0,0,0], [9E9, 9E9, 9E9, 9E9, 9E9, 9E9]];
	VAR robtarget OpenholeUD_5421 := [[377.32, -35.1, 172.38], [-0.183051, 0.683002, 0.683002, 0.183051], [0,0,0,0], [9E9, 9E9, 9E9, 9E9, 9E9, 9E9]];
	VAR robtarget OpenholeUD_5422 := [[381.32, -35.1, 172.36], [-0.183051, 0.683002, 0.683002, 0.183051], [0,0,0,0], [9E9, 9E9, 9E9, 9E9, 9E9, 9E9]];
	VAR robtarget OpenholeUD_5423 := [[385.32, -35.1, 172.35], [-0.183051, 0.683002, 0.683002, 0.183051], [0,0,0,0], [9E9, 9E9, 9E9, 9E9, 9E9, 9E9]];
	VAR robtarget OpenholeUD_5424 := [[389.32, -35.1, 172.34], [-0.136723, 0.693763, 0.669287, 0.228156], [0,0,0,0], [9E9, 9E9, 9E9, 9E9, 9E9, 9E9]];
	VAR robtarget OpenholeUD_5425 := [[393.27, -35.1, 172.95], [-0.12585, 0.695817, 0.672279, 0.219183], [0,0,0,0], [9E9, 9E9, 9E9, 9E9, 9E9, 9E9]];
	VAR robtarget OpenholeUD_5426 := [[397.22, -35.1, 173.56], [-0.114634, 0.697753, 0.675253, 0.209841], [0,0,0,0], [9E9, 9E9, 9E9, 9E9, 9E9, 9E9]];
	VAR robtarget OpenholeUD_5427 := [[401.18, -35.1, 174.17], [-0.103084, 0.699552, 0.678196, 0.200126], [0,0,0,0], [9E9, 9E9, 9E9, 9E9, 9E9, 9E9]];
	VAR robtarget OpenholeUD_5428 := [[405.13, -35.1, 174.78], [-0.091213, 0.701199, 0.681092, 0.190037], [0,0,0,0], [9E9, 9E9, 9E9, 9E9, 9E9, 9E9]];
	VAR robtarget OpenholeUD_5429 := [[409.08, -35.1, 175.4], [-0.079037, 0.702676, 0.683925, 0.179574], [0,0,0,0], [9E9, 9E9, 9E9, 9E9, 9E9, 9E9]];
	VAR robtarget OpenholeUD_5430 := [[413.04, -35.1, 176.01], [-0.066577, 0.703966, 0.686677, 0.168744], [0,0,0,0], [9E9, 9E9, 9E9, 9E9, 9E9, 9E9]];
	VAR robtarget OpenholeUD_5431 := [[416.99, -35.1, 176.62], [-0.053856, 0.705053, 0.689331, 0.157554], [0,0,0,0], [9E9, 9E9, 9E9, 9E9, 9E9, 9E9]];
	VAR robtarget OpenholeUD_5432 := [[420.94, -35.1, 177.23], [-0.040903, 0.705923, 0.691866, 0.146017], [0,0,0,0], [9E9, 9E9, 9E9, 9E9, 9E9, 9E9]];
	VAR robtarget OpenholeUD_5433 := [[424.89, -35.1, 177.84], [-0.027752, 0.706562, 0.694265, 0.134149], [0,0,0,0], [9E9, 9E9, 9E9, 9E9, 9E9, 9E9]];
	VAR robtarget OpenholeUD_5434 := [[428.85, -35.1, 178.45], [-0.014436, 0.706959, 0.696508, 0.121971], [0,0,0,0], [9E9, 9E9, 9E9, 9E9, 9E9, 9E9]];
	VAR robtarget OpenholeUD_5435 := [[432.8, -35.1, 179.06], [-0.000997, 0.707106, 0.698576, 0.109507], [0,0,0,0], [9E9, 9E9, 9E9, 9E9, 9E9, 9E9]];
	VAR robtarget OpenholeUD_5436 := [[436.75, -35.1, 179.67], [0.012525, 0.706996, 0.700452, 0.096786], [0,0,0,0], [9E9, 9E9, 9E9, 9E9, 9E9, 9E9]];
	VAR robtarget OpenholeUD_5437 := [[440.71, -35.1, 180.29], [0.026087, 0.706625, 0.702119, 0.083841], [0,0,0,0], [9E9, 9E9, 9E9, 9E9, 9E9, 9E9]];
	VAR robtarget OpenholeUD_5438 := [[444.66, -35.1, 180.9], [0.039642, 0.705995, 0.703563, 0.070708], [0,0,0,0], [9E9, 9E9, 9E9, 9E9, 9E9, 9E9]];
	VAR robtarget OpenholeUD_5439 := [[448.61, -35.1, 181.51], [0.053147, 0.705107, 0.704771, 0.057426], [0,0,0,0], [9E9, 9E9, 9E9, 9E9, 9E9, 9E9]];
	VAR robtarget OpenholeUD_5440 := [[452.57, -35.1, 182.12], [0.066557, 0.703967, 0.705734, 0.044036], [0,0,0,0], [9E9, 9E9, 9E9, 9E9, 9E9, 9E9]];
	VAR robtarget OpenholeUD_5441 := [[456.52, -35.1, 182.73], [0.079829, 0.702586, 0.706445, 0.030582], [0,0,0,0], [9E9, 9E9, 9E9, 9E9, 9E9, 9E9]];
	VAR robtarget OpenholeUD_5442 := [[460.47, -35.1, 183.34], [0.092921, 0.700975, 0.7069, 0.017107], [0,0,0,0], [9E9, 9E9, 9E9, 9E9, 9E9, 9E9]];
	VAR robtarget OpenholeUD_5443 := [[464.43, -35.1, 183.95], [0.105796, 0.699148, 0.707097, 0.003655], [0,0,0,0], [9E9, 9E9, 9E9, 9E9, 9E9, 9E9]];
	VAR robtarget OpenholeUD_5444 := [[468.38, -35.1, 184.56], [0.118419, 0.697121, 0.70704, -0.009732], [0,0,0,0], [9E9, 9E9, 9E9, 9E9, 9E9, 9E9]];
	VAR robtarget OpenholeUD_5445 := [[472.33, -35.1, 185.18], [0.130759, 0.694912, 0.706732, -0.023011], [0,0,0,0], [9E9, 9E9, 9E9, 9E9, 9E9, 9E9]];
	VAR robtarget OpenholeUD_5446 := [[476.28, -35.1, 185.79], [0.142789, 0.69254, 0.706182, -0.036144], [0,0,0,0], [9E9, 9E9, 9E9, 9E9, 9E9, 9E9]];
	VAR robtarget OpenholeUD_5447 := [[480.24, -35.1, 186.4], [0.154489, 0.690024, 0.7054, -0.049094], [0,0,0,0], [9E9, 9E9, 9E9, 9E9, 9E9, 9E9]];
	VAR robtarget OpenholeUD_5448 := [[484.19, -35.1, 187.01], [0.165839, 0.687385, 0.704398, -0.06183], [0,0,0,0], [9E9, 9E9, 9E9, 9E9, 9E9, 9E9]];
	VAR robtarget OpenholeUD_5449 := [[488.14, -35.1, 187.62], [0.176826, 0.68464, 0.70319, -0.07432], [0,0,0,0], [9E9, 9E9, 9E9, 9E9, 9E9, 9E9]];
	VAR robtarget OpenholeUD_5450 := [[492.1, -35.1, 188.23], [0.187441, 0.681811, 0.701791, -0.08654], [0,0,0,0], [9E9, 9E9, 9E9, 9E9, 9E9, 9E9]];
	VAR robtarget OpenholeUD_5451 := [[496.05, -35.1, 188.84], [0.197678, 0.678913, 0.700217, -0.098467], [0,0,0,0], [9E9, 9E9, 9E9, 9E9, 9E9, 9E9]];
	VAR robtarget OpenholeUD_5452 := [[500, -35.1, 189.45], [0.207535, 0.675965, 0.698485, -0.110086], [0,0,0,0], [9E9, 9E9, 9E9, 9E9, 9E9, 9E9]];
	VAR robtarget OpenholeUD_5453 := [[503.96, -35.1, 190.07], [0.217012, 0.672983, 0.696611, -0.12138], [0,0,0,0], [9E9, 9E9, 9E9, 9E9, 9E9, 9E9]];
	VAR robtarget OpenholeUD_5454 := [[509.38, -35.1, 190.9], [0.183051, 0.683002, 0.683002, -0.183051], [0,0,0,0], [9E9, 9E9, 9E9, 9E9, 9E9, 9E9]];
	VAR robtarget OpenholeUD_5455 := [[513.38, -35.1, 190.89], [0.183051, 0.683002, 0.683002, -0.183051], [0,0,0,0], [9E9, 9E9, 9E9, 9E9, 9E9, 9E9]];
	VAR robtarget OpenholeUD_5456 := [[517.38, -35.1, 190.88], [0.183051, 0.683002, 0.683002, -0.183051], [0,0,0,0], [9E9, 9E9, 9E9, 9E9, 9E9, 9E9]];
	VAR robtarget OpenholeUD_5457 := [[521.38, -35.1, 190.87], [0.183051, 0.683002, 0.683002, -0.183051], [0,0,0,0], [9E9, 9E9, 9E9, 9E9, 9E9, 9E9]];
	VAR robtarget OpenholeUD_5458 := [[525.38, -35.1, 190.85], [0.183051, 0.683002, 0.683002, -0.183051], [0,0,0,0], [9E9, 9E9, 9E9, 9E9, 9E9, 9E9]];
	VAR robtarget OpenholeUD_5459 := [[529.38, -35.1, 190.84], [0.183051, 0.683002, 0.683002, -0.183051], [0,0,0,0], [9E9, 9E9, 9E9, 9E9, 9E9, 9E9]];
	VAR robtarget OpenholeUD_5460 := [[529.38, -35.1, 190.84], [0.183051, 0.683002, 0.683002, -0.183051], [0,0,0,0], [9E9, 9E9, 9E9, 9E9, 9E9, 9E9]];
	VAR robtarget OpenholeUD_5461 := [[529.38, -36.3, 191.53], [0.183051, 0.683002, 0.683002, -0.183051], [0,0,0,0], [9E9, 9E9, 9E9, 9E9, 9E9, 9E9]];
	VAR robtarget OpenholeUD_5462 := [[525.38, -36.3, 191.55], [0.183051, 0.683002, 0.683002, -0.183051], [0,0,0,0], [9E9, 9E9, 9E9, 9E9, 9E9, 9E9]];
	VAR robtarget OpenholeUD_5463 := [[521.38, -36.3, 191.56], [0.183051, 0.683002, 0.683002, -0.183051], [0,0,0,0], [9E9, 9E9, 9E9, 9E9, 9E9, 9E9]];
	VAR robtarget OpenholeUD_5464 := [[517.38, -36.3, 191.57], [0.183051, 0.683002, 0.683002, -0.183051], [0,0,0,0], [9E9, 9E9, 9E9, 9E9, 9E9, 9E9]];
	VAR robtarget OpenholeUD_5465 := [[513.38, -36.3, 191.58], [0.183051, 0.683002, 0.683002, -0.183051], [0,0,0,0], [9E9, 9E9, 9E9, 9E9, 9E9, 9E9]];
	VAR robtarget OpenholeUD_5466 := [[509.38, -36.3, 191.6], [0.183051, 0.683002, 0.683002, -0.183051], [0,0,0,0], [9E9, 9E9, 9E9, 9E9, 9E9, 9E9]];
	VAR robtarget OpenholeUD_5467 := [[505.43, -36.3, 190.94], [0.2238, 0.670756, 0.696492, -0.122058], [0,0,0,0], [9E9, 9E9, 9E9, 9E9, 9E9, 9E9]];
	VAR robtarget OpenholeUD_5468 := [[501.49, -36.3, 190.29], [0.214547, 0.673773, 0.698364, -0.110847], [0,0,0,0], [9E9, 9E9, 9E9, 9E9, 9E9, 9E9]];
	VAR robtarget OpenholeUD_5469 := [[497.54, -36.3, 189.63], [0.204915, 0.676764, 0.700098, -0.099311], [0,0,0,0], [9E9, 9E9, 9E9, 9E9, 9E9, 9E9]];
	VAR robtarget OpenholeUD_5470 := [[493.6, -36.3, 188.97], [0.194903, 0.679715, 0.701677, -0.087463], [0,0,0,0], [9E9, 9E9, 9E9, 9E9, 9E9, 9E9]];
	VAR robtarget OpenholeUD_5471 := [[489.65, -36.3, 188.32], [0.184511, 0.682609, 0.703084, -0.07532], [0,0,0,0], [9E9, 9E9, 9E9, 9E9, 9E9, 9E9]];
	VAR robtarget OpenholeUD_5472 := [[485.7, -36.3, 187.66], [0.173743, 0.685429, 0.704303, -0.062903], [0,0,0,0], [9E9, 9E9, 9E9, 9E9, 9E9, 9E9]];
	VAR robtarget OpenholeUD_5473 := [[481.76, -36.3, 187.01], [0.162606, 0.688156, 0.70532, -0.050236], [0,0,0,0], [9E9, 9E9, 9E9, 9E9, 9E9, 9E9]];
	VAR robtarget OpenholeUD_5474 := [[477.81, -36.3, 186.35], [0.151112, 0.690772, 0.70612, -0.037347], [0,0,0,0], [9E9, 9E9, 9E9, 9E9, 9E9, 9E9]];
	VAR robtarget OpenholeUD_5475 := [[473.87, -36.3, 185.7], [0.139275, 0.693255, 0.70669, -0.024267], [0,0,0,0], [9E9, 9E9, 9E9, 9E9, 9E9, 9E9]];
